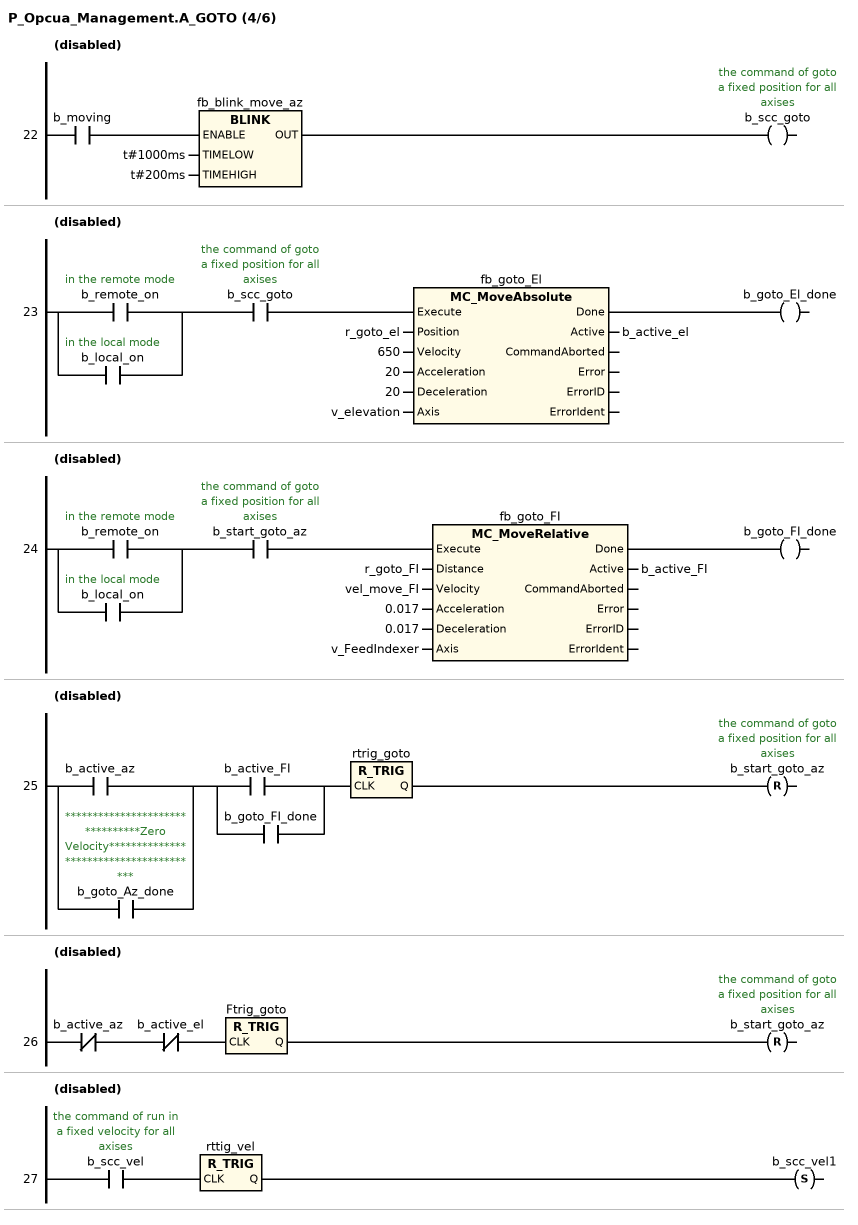
// NETWORK 22 (disabled)
//   b_scc_goto: the command of goto a fixed position for all axises
// fb_blink_move_az(ENABLE := b_moving, TIMELOW := t#1000ms, TIMEHIGH := t#200ms); // BLINK
// b_scc_goto := fb_blink_move_az.OUT;

// NETWORK 23 (disabled)
//   b_remote_on: in the remote mode
//   b_local_on: in the local mode
//   b_scc_goto: the command of goto a fixed position for all axises
//   v_elevation: Virtual axis "v_elevation" with axis number 8
// fb_goto_El(
//     Execute := (b_remote_on OR b_local_on) AND b_scc_goto,
//     Position := r_goto_el,
//     Velocity := 650,
//     Acceleration := 20,
//     Deceleration := 20,
//     Axis := v_elevation,
//     Active => b_active_el); // MC_MoveAbsolute
// b_goto_El_done := fb_goto_El.Done;

// NETWORK 24 (disabled)
//   b_remote_on: in the remote mode
//   b_local_on: in the local mode
//   b_start_goto_az: the command of goto a fixed position for all axises
//   v_FeedIndexer: Virtual axis "v_polarization" with axis number 9
// fb_goto_FI(
//     Execute := (b_remote_on OR b_local_on) AND b_start_goto_az,
//     Distance := r_goto_FI,
//     Velocity := vel_move_FI,
//     Acceleration := 0.017,
//     Deceleration := 0.017,
//     Axis := v_FeedIndexer,
//     Active => b_active_FI); // MC_MoveRelative
// b_goto_FI_done := fb_goto_FI.Done;

// NETWORK 25 (disabled)
//   b_goto_Az_done: ********************************Zero Velocity***************************************
//   b_start_goto_az: the command of goto a fixed position for all axises
// rtrig_goto(CLK := (b_active_az OR b_goto_Az_done) AND (b_active_FI OR b_goto_FI_done)); // R_TRIG
// b_start_goto_az R= rtrig_goto.Q;

// NETWORK 26 (disabled)
//   b_start_goto_az: the command of goto a fixed position for all axises
// Ftrig_goto(CLK := NOT b_active_az AND NOT b_active_el); // R_TRIG
// b_start_goto_az R= Ftrig_goto.Q;

// NETWORK 27 (disabled)
//   b_scc_vel: the command of run in a fixed velocity for all axises
// rttig_vel(CLK := b_scc_vel); // R_TRIG
// b_scc_vel1 S= rttig_vel.Q;

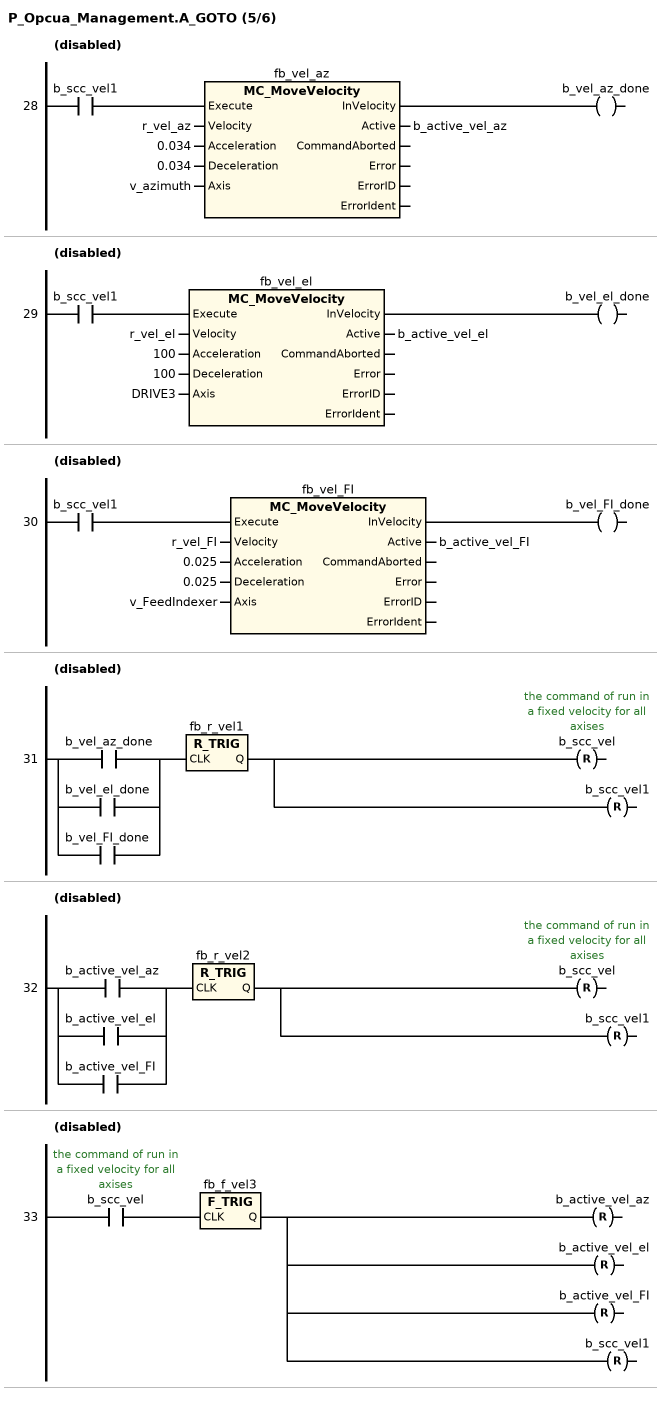
// NETWORK 28 (disabled)
//   r_vel_az: ************vel*************
//   v_azimuth: Virtual axis "v_azimuth" with axis number 7
// fb_vel_az(
//     Execute := b_scc_vel1,
//     Velocity := r_vel_az,
//     Acceleration := 0.034,
//     Deceleration := 0.034,
//     Axis := v_azimuth,
//     Active => b_active_vel_az); // MC_MoveVelocity
// b_vel_az_done := fb_vel_az.InVelocity;

// NETWORK 29 (disabled)
//   DRIVE3: Virtual axis "v_elevation" with axis number 8
// fb_vel_el(
//     Execute := b_scc_vel1,
//     Velocity := r_vel_el,
//     Acceleration := 100,
//     Deceleration := 100,
//     Axis := DRIVE3,
//     Active => b_active_vel_el); // MC_MoveVelocity
// b_vel_el_done := fb_vel_el.InVelocity;

// NETWORK 30 (disabled)
//   v_FeedIndexer: Virtual axis "v_polarization" with axis number 9
// fb_vel_FI(
//     Execute := b_scc_vel1,
//     Velocity := r_vel_FI,
//     Acceleration := 0.025,
//     Deceleration := 0.025,
//     Axis := v_FeedIndexer,
//     Active => b_active_vel_FI); // MC_MoveVelocity
// b_vel_FI_done := fb_vel_FI.InVelocity;

// NETWORK 31 (disabled)
//   b_scc_vel: the command of run in a fixed velocity for all axises
// fb_r_vel1(CLK := b_vel_az_done OR b_vel_el_done OR b_vel_FI_done); // R_TRIG
// b_scc_vel R= fb_r_vel1.Q;
// b_scc_vel1 R= fb_r_vel1.Q;

// NETWORK 32 (disabled)
//   b_scc_vel: the command of run in a fixed velocity for all axises
// fb_r_vel2(CLK := b_active_vel_az OR b_active_vel_el OR b_active_vel_FI); // R_TRIG
// b_scc_vel R= fb_r_vel2.Q;
// b_scc_vel1 R= fb_r_vel2.Q;

// NETWORK 33 (disabled)
//   b_scc_vel: the command of run in a fixed velocity for all axises
// fb_f_vel3(CLK := b_scc_vel); // F_TRIG
// b_active_vel_az R= fb_f_vel3.Q;
// b_active_vel_el R= fb_f_vel3.Q;
// b_active_vel_FI R= fb_f_vel3.Q;
// b_scc_vel1 R= fb_f_vel3.Q;

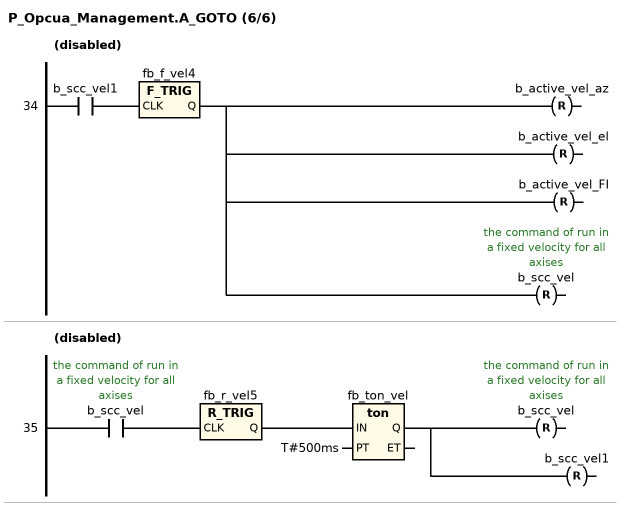
// NETWORK 34 (disabled)
//   b_scc_vel: the command of run in a fixed velocity for all axises
// fb_f_vel4(CLK := b_scc_vel1); // F_TRIG
// b_active_vel_az R= fb_f_vel4.Q;
// b_active_vel_el R= fb_f_vel4.Q;
// b_active_vel_FI R= fb_f_vel4.Q;
// b_scc_vel R= fb_f_vel4.Q;

// NETWORK 35 (disabled)
//   b_scc_vel: the command of run in a fixed velocity for all axises
// fb_r_vel5(CLK := b_scc_vel); // R_TRIG
// fb_ton_vel(IN := fb_r_vel5.Q, PT := T#500ms); // ton
// b_scc_vel R= fb_ton_vel.Q;
// b_scc_vel1 R= fb_ton_vel.Q;
END_ACTION

ACTION A_CLR_ERR:
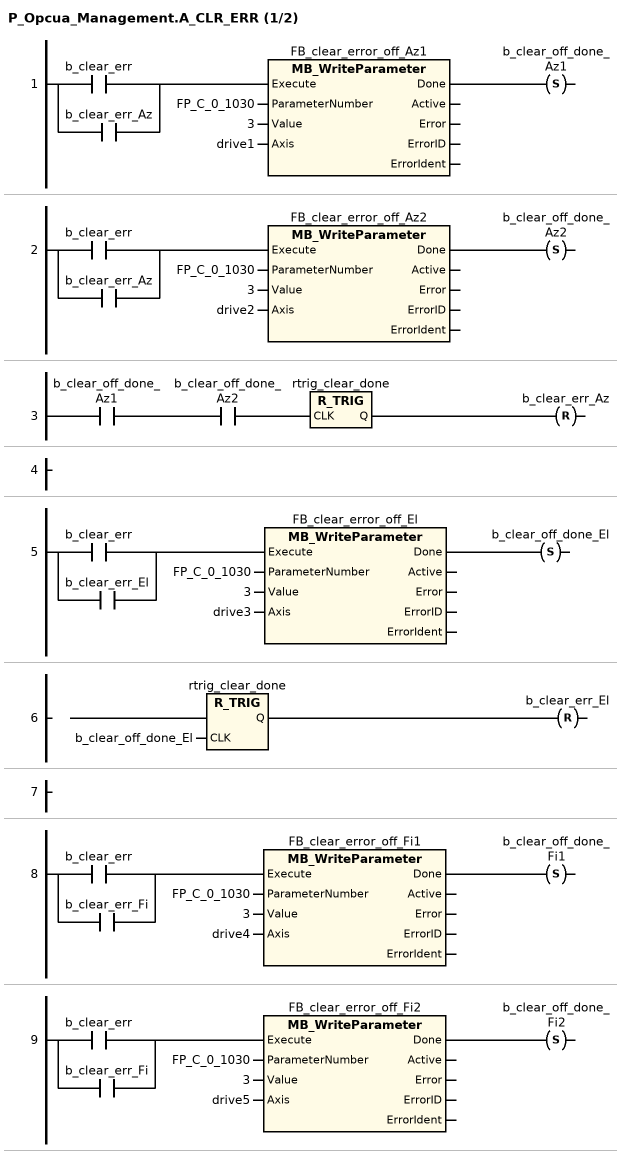
// NETWORK 1
//   FP_C_0_1030: Command: Clear all control errors
//   drive1: Real axis "Drive1" with axis number 1
FB_clear_error_off_Az1(
    Execute := b_clear_err OR b_clear_err_Az,
    ParameterNumber := FP_C_0_1030,
    Value := 3,
    Axis := drive1); // MB_WriteParameter
b_clear_off_done_Az1 S= FB_clear_error_off_Az1.Done;

// NETWORK 2
//   FP_C_0_1030: Command: Clear all control errors
//   drive2: Real axis "Drive1" with axis number 1
FB_clear_error_off_Az2(
    Execute := b_clear_err OR b_clear_err_Az,
    ParameterNumber := FP_C_0_1030,
    Value := 3,
    Axis := drive2); // MB_WriteParameter
b_clear_off_done_Az2 S= FB_clear_error_off_Az2.Done;

// NETWORK 3
rtrig_clear_done(CLK := b_clear_off_done_Az1 AND b_clear_off_done_Az2); // R_TRIG
b_clear_err_Az R= rtrig_clear_done.Q;

// NETWORK 4

// NETWORK 5
//   FP_C_0_1030: Command: Clear all control errors
//   drive3: Real axis "Drive1" with axis number 1
FB_clear_error_off_El(
    Execute := b_clear_err OR b_clear_err_El,
    ParameterNumber := FP_C_0_1030,
    Value := 3,
    Axis := drive3); // MB_WriteParameter
b_clear_off_done_El S= FB_clear_error_off_El.Done;

// NETWORK 6
rtrig_clear_done(CLK := b_clear_off_done_El); // R_TRIG
b_clear_err_El R= rtrig_clear_done.Q;

// NETWORK 7

// NETWORK 8
//   FP_C_0_1030: Command: Clear all control errors
//   drive4: Real axis "Drive1" with axis number 1
FB_clear_error_off_Fi1(
    Execute := b_clear_err OR b_clear_err_Fi,
    ParameterNumber := FP_C_0_1030,
    Value := 3,
    Axis := drive4); // MB_WriteParameter
b_clear_off_done_Fi1 S= FB_clear_error_off_Fi1.Done;

// NETWORK 9
//   FP_C_0_1030: Command: Clear all control errors
//   drive5: Real axis "Drive1" with axis number 1
FB_clear_error_off_Fi2(
    Execute := b_clear_err OR b_clear_err_Fi,
    ParameterNumber := FP_C_0_1030,
    Value := 3,
    Axis := drive5); // MB_WriteParameter
b_clear_off_done_Fi2 S= FB_clear_error_off_Fi2.Done;

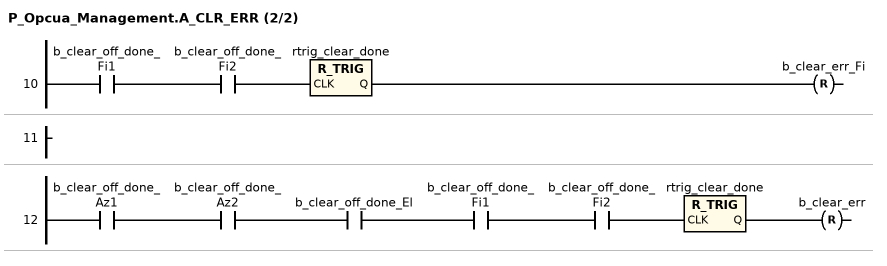
// NETWORK 10
rtrig_clear_done(CLK := b_clear_off_done_Fi1 AND b_clear_off_done_Fi2); // R_TRIG
b_clear_err_Fi R= rtrig_clear_done.Q;

// NETWORK 11

// NETWORK 12
rtrig_clear_done(CLK := b_clear_off_done_Az1 AND b_clear_off_done_Az2 AND b_clear_off_done_El AND b_clear_off_done_Fi1 AND b_clear_off_done_Fi2); // R_TRIG
b_clear_err R= rtrig_clear_done.Q;
END_ACTION

END_PROGRAM

// IndraMotionMlc1/Application/POUs/OPCUA/OPCUA_Node/P_Opcua_Tracking
{attribute 'linkalways'}
PROGRAM P_Opcua_Tracking
VAR_INPUT
	
	i_length: UINT;
	tai: ARRAY [1..1000] OF LREAL;
	Az: ARRAY [1..1000] OF LREAL;
	El: ARRAY [1..1000] OF LREAL;
	
END_VAR

VAR
	index: UINT; // Index used for addressing points in the tracking data arrays. 
	
	IL_LowPass_OnSource: IL_StateVariableType01;
	b_test: BOOL;
	
END_VAR


// Switch track on if the starttime has been reached
IF b_track_start AND (lr_track_start_time <= Time_cds.Status.TAIoffset) THEN 
	b_track_on:=1;
	b_track_start:=0;
END_IF

//IF i_length>0 THEN  // Load table into stack 
	
	
//END_IF

// Calculate whether the dish is on source. 

IF b_track_on THEN 
	IF  tracking.status.OnSourceDev <= Tracking.Status.OnSourceThreshold THEN 
		Management.Status.OnSource:=1;
	ELSE
		Management.Status.OnSource:=0;	
	END_IF
ELSE
	Management.Status.OnSource:=0;
END_IF

//Tracking.Status.act_statOffset_value_El  Updated in P_Track_cubic
//Tracking.Status.act_statOffset_value_Xel Updated in P_Track_cubic
//Tracking.Status.OnSourceDev              Updated in P_Track_cubic
//Tracking.Status.OnSourceThreshold        Updated in SetOnSourceThreshold
//Tracking.Status.p_desired_Az;            Updated in P_Track_cubic
//Tracking.Status.p_desired_El;            Updated in P_Track_cubic
//Tracking.Status.ThresholdTimePeriod      Updated in SetOnSourceThreshold
IF Management.Status.DscState=DscStatetype.Standby OR Management.Status.DscState=DscStatetype.Standstill OR Management.Status.DscState=DscStatetype.Slew OR Management.Status.DscState=DscStatetype.Track THEN 
	Tracking.Status.tr_initOk:=1;
ELSE 
	Tracking.Status.tr_initOk:=0;
END_IF

Tracking.Status.tr_obj_valid:= Tracking.TableStatus.pts_DataValid;
Tracking.Status.tr_selPoly:= 0;

IF Tracking.TableStatus.pts_DataValid THEN
	Tracking.Status.tr_TimeRemaining:= ABS(track_table[i_End].TAIoffset - track_table[i_Start].TAIoffset);
ELSE
	Tracking.Status.tr_TimeRemaining:=0;
END_IF

IF (track_table[i_End].TAIoffset)>(Time_cds.Status.TAIoffset+600) THEN  // Minimum of 10min track data available . 
	Tracking.Status.tr_valid:=1;
ELSE
	Tracking.Status.tr_valid:=0;
END_IF

Tracking.TableStatus.act_pt_act_index := INT_TO_UINT(i_Start);
Tracking.TableStatus.act_pt_end_index := INT_TO_UINT(i_End);
Tracking.TableStatus.act_pt_value_Az:= track_table[i_Start].Azimuth;
Tracking.TableStatus.act_pt_value_El:= track_table[i_Start].Elevation;
//Tracking.TableStatus.LastLoadMode; Updated in TrackloadTable
IF i_num_stack_left > 10 THEN
	Tracking.TableStatus.pts_Completed:=0; 
	ELSE
	Tracking.TableStatus.pts_Completed:=1;
END_IF
IF Tracking.TableStatus.pts_Completed THEN 
	Tracking.TableStatus.pts_DataValid:=0; // Once a track is finnished then there is no valid data to trck with. 
END_IF
Tracking.TableStatus.pts_Err:=0; 
//Tracking.TableStatus.pts_Interpol;  Updated in Track Start
Tracking.TableStatus.pts_InterpolError:=0;  // Don't have code for detecting interpolaor errors yet
Tracking.TableStatus.pts_Running:=b_track_on;
Tracking.TableStatus.pts_StartPos:=b_track_on;

IF i_num_stack_left<=60 AND i_num_stack_left >= 70 THEN
	Tracking.TableStatus.pts_TableAlmostFull:=1;
ELSE 
	Tracking.TableStatus.pts_TableAlmostFull:=0;
END_IF

P_Opcua_Tracking.A_Utils();

ACTION A_Utils:
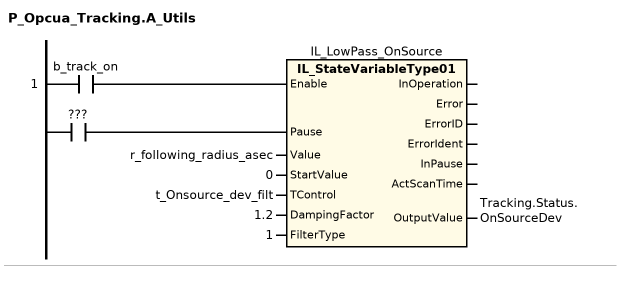
// NETWORK 1
IL_LowPass_OnSource(
    Enable := b_track_on,
    Value := r_following_radius_asec,
    StartValue := 0,
    TControl := t_Onsource_dev_filt,
    DampingFactor := 1.2,
    FilterType := 1,
    OutputValue => Tracking.Status.OnSourceDev); // IL_StateVariableType01
END_ACTION

END_PROGRAM

// IndraMotionMlc1/Application/POUs/OPCUA/OPCUA_Node/P_Opcua_Pointing
PROGRAM P_Opcua_Pointing
VAR
	TiltTemp_mV_1: LREAL;
	lr_one_x_off: LREAL;
	lr_one_y_off: LREAL;
	TiltTemp_mV_2: LREAL;
	lr_two_x_off: LREAL;
	lr_two_y_off: LREAL;
	IL_LowPass_Tilt_one_x: IL_StateVariableType01;
	IL_LowPass_Tilt_one_y: IL_StateVariableType01;
	IL_LowPass_Tilt_two_x: IL_StateVariableType01;
	IL_LowPass_Tilt_two_y: IL_StateVariableType01;
	t_one_x_filt_dt: TIME;
	t_one_y_filt_dt: TIME;
	t_two_x_filt_dt: TIME;
	t_two_y_filt_dt: TIME;
	b_tilt_filt_on: BOOL:= 1;
	RunOnce:Bool:=True;
END_VAR

Pointing();
(*****Data*****)
IF RunOnce THEN
	Pointing.StaticPmParameters:=StaticPmParametersSave;
	Pointing.TiltmeterParameters:=TiltmeterParametersSave;
	Pointing.AmbTempParameters:= AmbTempParametersSave;
	RunOnce:=FALSE; 
END_IF

(****************** Tilt Sensor **************************************)
// Tilt sensor one
Pointing.Status.TiltTemp_One := TiltTemp_mV_1*0.1;

lr_one_x_off:= (Pointing.TiltmeterParameters.One.x_zero+Pointing.TiltmeterParameters.One.x_zeroTC*Pointing.Status.TiltTemp_One)+
(Pointing.TiltmeterParameters.One.x_off+Pointing.TiltmeterParameters.One.x_offTC*Pointing.Status.TiltTemp_One);
lr_one_y_off:=(Pointing.TiltmeterParameters.One.y_zero+Pointing.TiltmeterParameters.One.y_zeroTC*Pointing.Status.TiltTemp_One)+
(Pointing.TiltmeterParameters.One.y_off+Pointing.TiltmeterParameters.One.y_offTC*Pointing.Status.TiltTemp_One);

Pointing.Status.TiltXArcsec_One:= Pointing.Status.TiltXRaw_mV_One*(Pointing.TiltmeterParameters.One.x_scale+Pointing.TiltmeterParameters.One.x_scaleTC*Pointing.Status.TiltTemp_One)+Pointing.TiltmeterParameters.One.x_off;
Pointing.Status.TiltYArcsec_One:= Pointing.Status.TiltYRaw_mV_One*(Pointing.TiltmeterParameters.One.y_scale+Pointing.TiltmeterParameters.One.y_scaleTC*Pointing.Status.TiltTemp_One)+Pointing.TiltmeterParameters.One.y_off;
t_one_x_filt_dt:= TO_TIME(Pointing.TiltmeterParameters.One.x_filt_dt*1000); //convert to milliseconds and TIME type.
t_one_y_filt_dt:= TO_TIME(Pointing.TiltmeterParameters.One.y_filt_dt*1000);

// Tilt Sensor Two
Pointing.Status.TiltTemp_Two := TiltTemp_mV_2*0.1;

lr_two_x_off:= (Pointing.TiltmeterParameters.Two.x_zero+Pointing.TiltmeterParameters.Two.x_zeroTC*Pointing.Status.TiltTemp_Two)+
(Pointing.TiltmeterParameters.Two.x_off+Pointing.TiltmeterParameters.Two.x_offTC*Pointing.Status.TiltTemp_Two);
lr_two_y_off:=(Pointing.TiltmeterParameters.Two.y_zero+Pointing.TiltmeterParameters.Two.y_zeroTC*Pointing.Status.TiltTemp_Two)+
(Pointing.TiltmeterParameters.Two.y_off+Pointing.TiltmeterParameters.Two.y_offTC*Pointing.Status.TiltTemp_Two);

Pointing.Status.TiltXArcsec_Two:= Pointing.Status.TiltXRaw_mV_Two*(Pointing.TiltmeterParameters.Two.x_scale+Pointing.TiltmeterParameters.Two.x_scaleTC*Pointing.Status.TiltTemp_Two)+Pointing.TiltmeterParameters.Two.x_off;
Pointing.Status.TiltYArcsec_Two:= Pointing.Status.TiltYRaw_mV_Two*(Pointing.TiltmeterParameters.Two.y_scale+Pointing.TiltmeterParameters.Two.y_scaleTC*Pointing.Status.TiltTemp_Two)+Pointing.TiltmeterParameters.Two.y_off;
t_two_x_filt_dt:= TO_TIME(Pointing.TiltmeterParameters.Two.x_filt_dt*1000); //convert to milliseconds and TIME type.
t_two_y_filt_dt:= TO_TIME(Pointing.TiltmeterParameters.Two.y_filt_dt*1000);

// Total point corrections

Pointing.Status.TotalPointCorr_Az:= Pointing.Status.StaticPmCorrVal_Az + Pointing.Status.TiltCorrVal_Az + Pointing.Status.AmbTempCorrVal_Az;
Pointing.Status.TotalPointCorr_El:= Pointing.Status.StaticPmCorrVal_El + Pointing.Status.TiltCorrVal_El + Pointing.Status.AmbTempCorrVal_El;

Pointing.Status.ActAmbTemp_East:= Pedestal_temp_1;  // These need to be checked
Pointing.Status.ActAmbTemp_South:= Pedestal_temp_2;;
Pointing.Status.ActAmbTemp_West:= Pedestal_temp_3;
//Pointing.Status.AmbTempCorrActive
//Pointing.Status.AmbTempCorrVal_Az
//Pointing.Status.AmbTempCorrVal_El
//Pointing.Status.BandForCorr
//Pointing.Status.StaticCorrActive
//Pointing.Status.StaticPmCorrVal_Az
//Pointing.Status.StaticPmCorrVal_El
//Pointing.Status.TiltCorrActive
//Pointing.Status.TiltCorrVal_Az
//Pointing.Status.TiltCorrVal_El
//Pointing.Status.TiltOne_On
//Pointing.Status.TiltTemp_One
//Pointing.Status.TiltTemp_Two
//Pointing.Status.TotalPointCorr_Az
//Pointing.Status.TotalPointCorr_El

ACTION A_Utils:
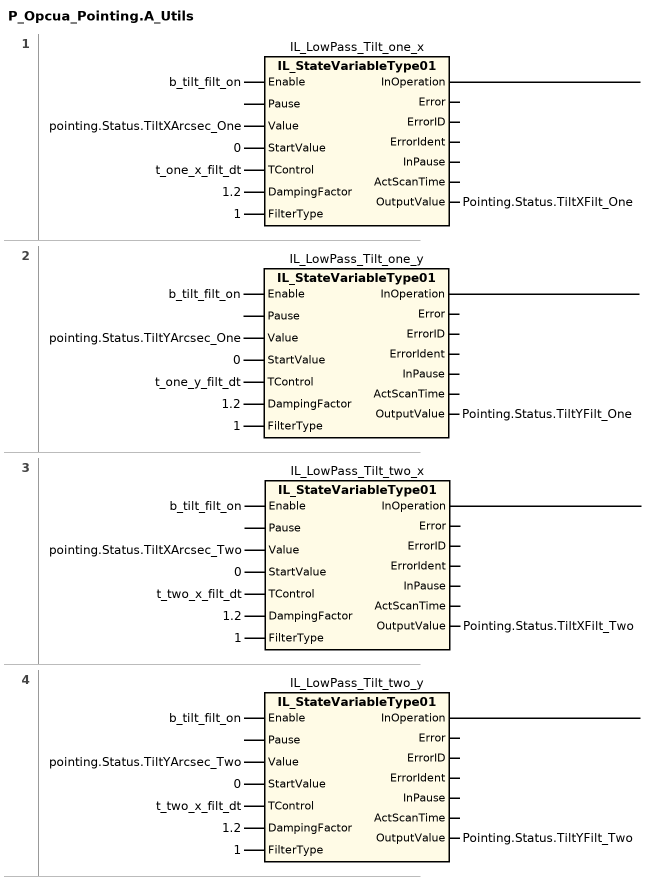
// NETWORK 1
IL_LowPass_Tilt_one_x(
    Enable := b_tilt_filt_on,
    Value := pointing.Status.TiltXArcsec_One,
    StartValue := 0,
    TControl := t_one_x_filt_dt,
    DampingFactor := 1.2,
    FilterType := 1,
    OutputValue => Pointing.Status.TiltXFilt_One); // IL_StateVariableType01

// NETWORK 2
IL_LowPass_Tilt_one_y(
    Enable := b_tilt_filt_on,
    Value := pointing.Status.TiltYArcsec_One,
    StartValue := 0,
    TControl := t_one_y_filt_dt,
    DampingFactor := 1.2,
    FilterType := 1,
    OutputValue => Pointing.Status.TiltYFilt_One); // IL_StateVariableType01

// NETWORK 3
IL_LowPass_Tilt_two_x(
    Enable := b_tilt_filt_on,
    Value := pointing.Status.TiltXArcsec_Two,
    StartValue := 0,
    TControl := t_two_x_filt_dt,
    DampingFactor := 1.2,
    FilterType := 1,
    OutputValue => Pointing.Status.TiltXFilt_Two); // IL_StateVariableType01

// NETWORK 4
IL_LowPass_Tilt_two_y(
    Enable := b_tilt_filt_on,
    Value := pointing.Status.TiltYArcsec_Two,
    StartValue := 0,
    TControl := t_two_x_filt_dt,
    DampingFactor := 1.2,
    FilterType := 1,
    OutputValue => Pointing.Status.TiltYFilt_Two); // IL_StateVariableType01
END_ACTION

END_PROGRAM

// IndraMotionMlc1/Application/POUs/Motion/Test_move
PROGRAM Test_move
VAR
	b_power: BOOL;
	b_enable_az1: BOOL;
	fb_enable_az1: MC_Power;
	b_enable_az1_done: BOOL;
	b_vel_az1: BOOL;
	fb_vel_az1: MC_MoveVelocity;
	vel_az1: REAL;
	b_enable_az2: BOOL;
	fb_enable_az2: MC_Power;
	b_enable_az2_done: BOOL;
	b_vel_az2: BOOL;
	vel_az2: REAL;
	fb_vel_az2: MC_MoveVelocity;
	b_enable_el1: BOOL;
	fb_enable_el1: MC_Power;
	b_enable_el1_done: BOOL;
	b_vel_el1: BOOL;
	vel_el1: REAL;
	fb_vel_el1: MC_MoveVelocity;
	b_vel_el2: BOOL;
	fb_vel_el2: MC_MoveVelocity;
	vel_el2: REAL;
	b_enable_el2: BOOL;
	fb_enable_el2: MC_Power;
	b_enable_FI1: BOOL;
	fb_enable_FI1: MC_Power;
	b_enable_el2_done: BOOL;
	b_enable_FI1_done: BOOL;
	b_vel_FI1: BOOL;
	fb_vel_FI1: MC_MoveVelocity;
	vel_FI1: REAL;
	b_enable_FI2: BOOL;
	fb_enable_FI2: MC_Power;
	b_enable_FI2_done: BOOL;
	b_vel_FI2: BOOL;
	vel_FI2: REAL;
	fb_vel_FI2: MC_MoveVelocity;
	b_torque_4: BOOL;
	b_torque_el2: BOOL;
	fb_torque_el2: MC_TorqueControl;
	b_torque_el2_done: BOOL;
	b_torque_az2: BOOL;
	fb_torque_az2: MC_TorqueControl;
	b_torque_az2_done: BOOL;
	fb_pos_az1: MC_MoveAbsolute;
	b_pos_az1: BOOL;
	pos_az1: REAL;
	b_stop_az: BOOL;
	fb_stop_AZ: MC_Stop;
	b_stop_el: BOOL;
	fb_stop_el: MC_Stop;
	b_pos_el1: BOOL;
	pos_el1: REAL;
	fb_pos_el1: MC_MoveAbsolute;
	b_pos_FI1: BOOL;
	pos_FI1: REAL;
	fb_pos_FI1: MC_MoveAbsolute;
	b_vel_1: BOOL;
	vel_1: REAL;
	fb_vel_1: MC_MoveVelocity;
	test_home_1: BOOL;
	fb_test_home: MB_Home;
	b_homeswitch_1: BOOL;
	b_torque_FI2: BOOL;
	fb_torque_FI2: MC_TorqueControl;
	b_torque_FI2_done: BOOL;
	b_touque_1: BOOL;
	fb_torque_az1: MC_TorqueControl;
	b_torque_az1_done: BOOL;
	torque_1: REAL;
	b_touque_3: BOOL;
	torque_3: REAL;
	fb_torque_el3: MC_TorqueControl;
END_VAR

(*IF r_pos_az>270.5 OR  r_pos_az<-270.5 THEN
			b_SCC_enable_on:=FALSE;
			b_SCC_enable_off:=TRUE; 
END_IF
*)




//axisdata[7].rActualPosition_i;
//test_move.power_move(); Commented out to prevent process using up resources.

ACTION power_move:
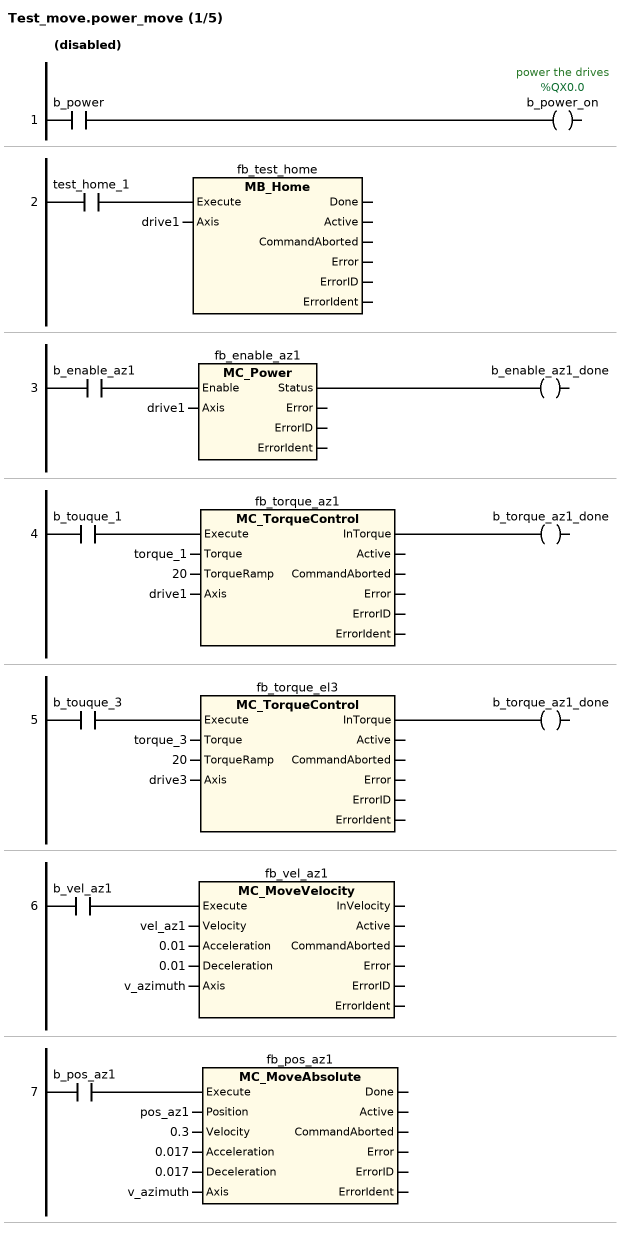
// NETWORK 1 (disabled)
//   b_power_on: power the drives | AT %QX0.0
// b_power_on := b_power;

// NETWORK 2
//   drive1: Real axis "Drive1" with axis number 1
fb_test_home(Execute := test_home_1, Axis := drive1); // MB_Home

// NETWORK 3
//   drive1: Real axis "Drive1" with axis number 1
fb_enable_az1(Enable := b_enable_az1, Axis := drive1); // MC_Power
b_enable_az1_done := fb_enable_az1.Status;

// NETWORK 4
//   drive1: Real axis "Drive4" with axis number 4
fb_torque_az1(Execute := b_touque_1, Torque := torque_1, TorqueRamp := 20, Axis := drive1); // MC_TorqueControl
b_torque_az1_done := fb_torque_az1.InTorque;

// NETWORK 5
//   drive3: Real axis "Drive4" with axis number 4
fb_torque_el3(Execute := b_touque_3, Torque := torque_3, TorqueRamp := 20, Axis := drive3); // MC_TorqueControl
b_torque_az1_done := fb_torque_el3.InTorque;

// NETWORK 6
//   v_azimuth: Virtual axis "v_azimuth" with axis number 7
fb_vel_az1(
    Execute := b_vel_az1,
    Velocity := vel_az1,
    Acceleration := 0.01,
    Deceleration := 0.01,
    Axis := v_azimuth); // MC_MoveVelocity

// NETWORK 7
//   v_azimuth: Virtual axis "v_azimuth" with axis number 7
fb_pos_az1(
    Execute := b_pos_az1,
    Position := pos_az1,
    Velocity := 0.3,
    Acceleration := 0.017,
    Deceleration := 0.017,
    Axis := v_azimuth); // MC_MoveAbsolute

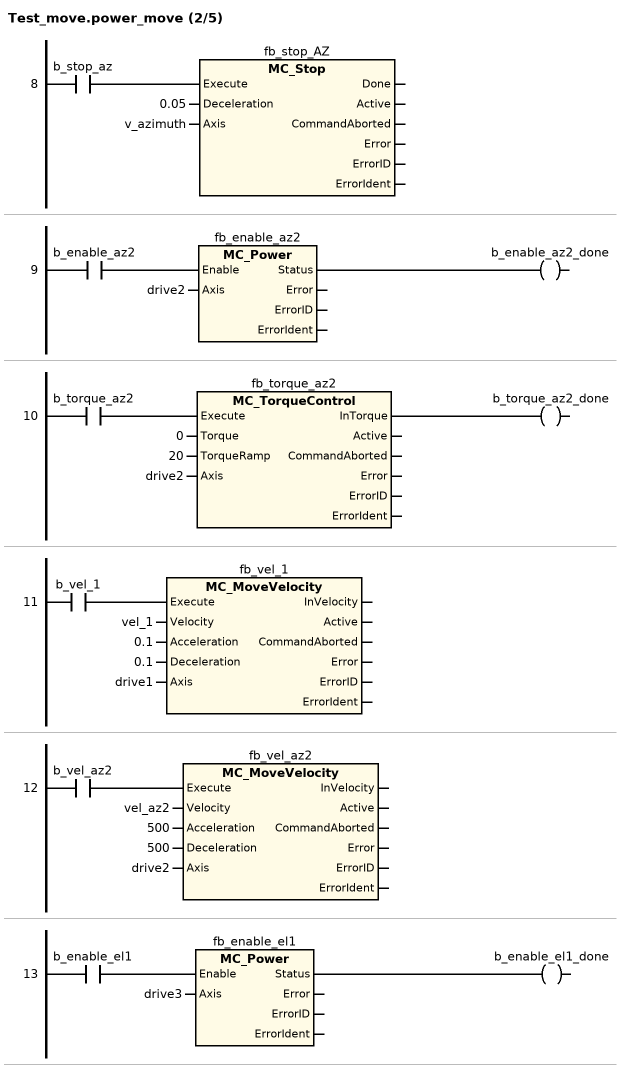
// NETWORK 8
//   v_azimuth: Virtual axis "v_azimuth" with axis number 7
fb_stop_AZ(Execute := b_stop_az, Deceleration := 0.05, Axis := v_azimuth); // MC_Stop

// NETWORK 9
//   drive2: Real axis "Drive2" with axis number 2
fb_enable_az2(Enable := b_enable_az2, Axis := drive2); // MC_Power
b_enable_az2_done := fb_enable_az2.Status;

// NETWORK 10
//   drive2: Real axis "Drive2" with axis number 2
fb_torque_az2(Execute := b_torque_az2, Torque := 0, TorqueRamp := 20, Axis := drive2); // MC_TorqueControl
b_torque_az2_done := fb_torque_az2.InTorque;

// NETWORK 11
//   drive1: Real axis "Drive1" with axis number 1
fb_vel_1(Execute := b_vel_1, Velocity := vel_1, Acceleration := 0.1, Deceleration := 0.1, Axis := drive1); // MC_MoveVelocity

// NETWORK 12
//   drive2: Real axis "Drive2" with axis number 2
fb_vel_az2(
    Execute := b_vel_az2,
    Velocity := vel_az2,
    Acceleration := 500,
    Deceleration := 500,
    Axis := drive2); // MC_MoveVelocity

// NETWORK 13
//   drive3: Real axis "Drive3" with axis number 3
fb_enable_el1(Enable := b_enable_el1, Axis := drive3); // MC_Power
b_enable_el1_done := fb_enable_el1.Status;

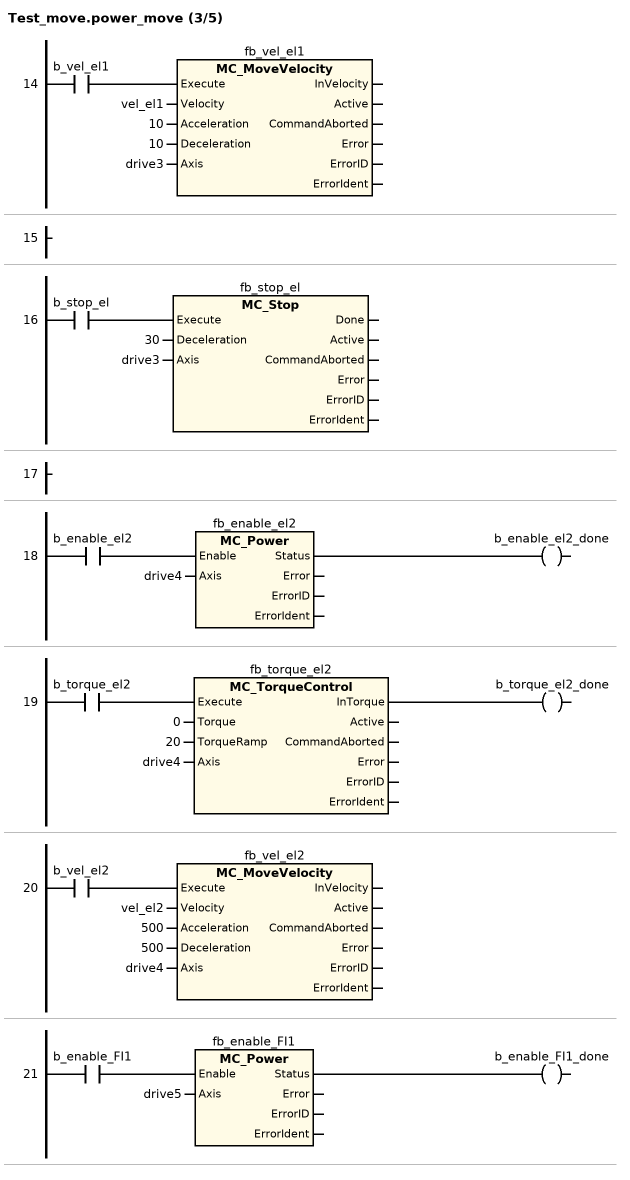
// NETWORK 14
//   drive3: Virtual axis "v_elevation" with axis number 8
fb_vel_el1(Execute := b_vel_el1, Velocity := vel_el1, Acceleration := 10, Deceleration := 10, Axis := drive3); // MC_MoveVelocity

// NETWORK 15

// NETWORK 16
//   drive3: Virtual axis "v_elevation" with axis number 8
fb_stop_el(Execute := b_stop_el, Deceleration := 30, Axis := drive3); // MC_Stop

// NETWORK 17

// NETWORK 18
//   drive4: Real axis "Drive4" with axis number 4
fb_enable_el2(Enable := b_enable_el2, Axis := drive4); // MC_Power
b_enable_el2_done := fb_enable_el2.Status;

// NETWORK 19
//   drive4: Real axis "Drive4" with axis number 4
fb_torque_el2(Execute := b_torque_el2, Torque := 0, TorqueRamp := 20, Axis := drive4); // MC_TorqueControl
b_torque_el2_done := fb_torque_el2.InTorque;

// NETWORK 20
//   drive4: Real axis "Drive4" with axis number 4
fb_vel_el2(
    Execute := b_vel_el2,
    Velocity := vel_el2,
    Acceleration := 500,
    Deceleration := 500,
    Axis := drive4); // MC_MoveVelocity

// NETWORK 21
//   drive5: Real axis "Drive5" with axis number 5
fb_enable_FI1(Enable := b_enable_FI1, Axis := drive5); // MC_Power
b_enable_FI1_done := fb_enable_FI1.Status;

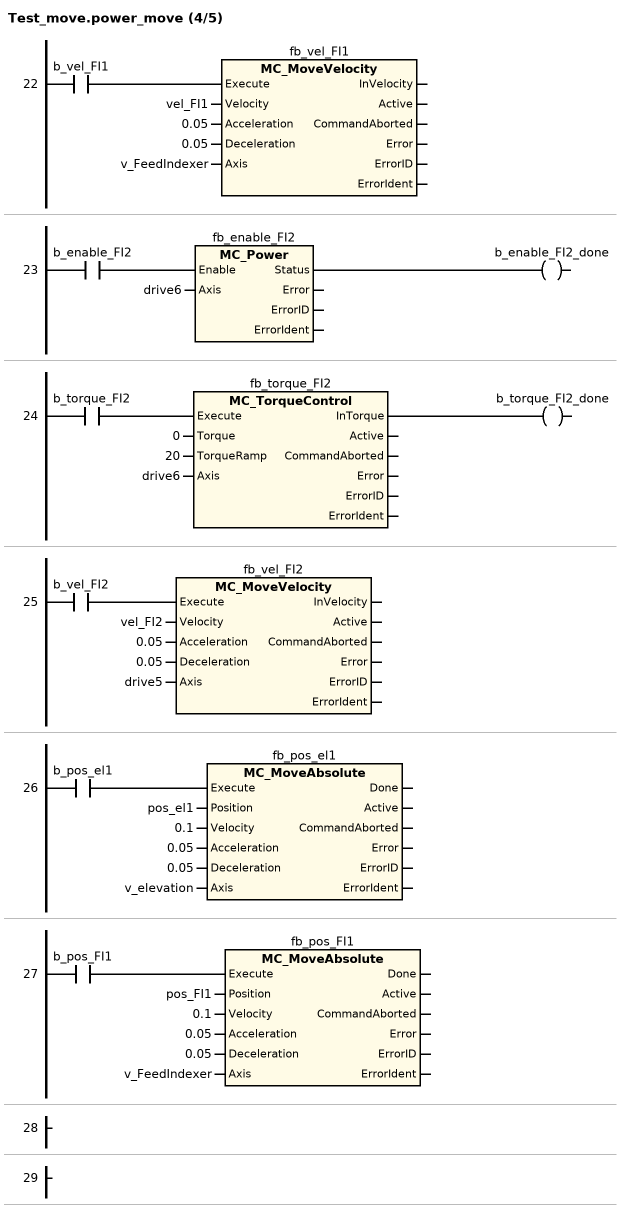
// NETWORK 22
//   v_FeedIndexer: Virtual axis "v_polarization" with axis number 9
fb_vel_FI1(
    Execute := b_vel_FI1,
    Velocity := vel_FI1,
    Acceleration := 0.05,
    Deceleration := 0.05,
    Axis := v_FeedIndexer); // MC_MoveVelocity

// NETWORK 23
//   drive6: Real axis "Drive6" with axis number 6
fb_enable_FI2(Enable := b_enable_FI2, Axis := drive6); // MC_Power
b_enable_FI2_done := fb_enable_FI2.Status;

// NETWORK 24
//   drive6: Real axis "Drive6" with axis number 6
fb_torque_FI2(Execute := b_torque_FI2, Torque := 0, TorqueRamp := 20, Axis := drive6); // MC_TorqueControl
b_torque_FI2_done := fb_torque_FI2.InTorque;

// NETWORK 25
//   drive5: Real axis "Drive5" with axis number 5
fb_vel_FI2(
    Execute := b_vel_FI2,
    Velocity := vel_FI2,
    Acceleration := 0.05,
    Deceleration := 0.05,
    Axis := drive5); // MC_MoveVelocity

// NETWORK 26
//   v_elevation: Virtual axis "v_elevation" with axis number 8
fb_pos_el1(
    Execute := b_pos_el1,
    Position := pos_el1,
    Velocity := 0.1,
    Acceleration := 0.05,
    Deceleration := 0.05,
    Axis := v_elevation); // MC_MoveAbsolute

// NETWORK 27
//   v_FeedIndexer: Virtual axis "v_polarization" with axis number 9
fb_pos_FI1(
    Execute := b_pos_FI1,
    Position := pos_FI1,
    Velocity := 0.1,
    Acceleration := 0.05,
    Deceleration := 0.05,
    Axis := v_FeedIndexer); // MC_MoveAbsolute

// NETWORK 28

// NETWORK 29

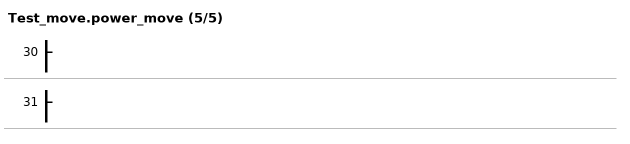
// NETWORK 30

// NETWORK 31
END_ACTION

END_PROGRAM

// IndraMotionMlc1/Application/POUs/Motion/PlcProg
PROGRAM PlcProg
VAR
	bVM_Enable: BOOL;
	rVM_Acc: REAL:=10.0;
	rVM_Dec: REAL:=10.0;
	rVM_Velocity: REAL:=3.0;
  rPhaseShift: REAL:=99.0;
	bVM_VelModeAck: BOOL;
	bVM_Standstill: BOOL;
	rVM_actVelocity: REAL;
END_VAR

//------------------------------------------------------------------------------------------------------
//--------------------- Call all required programs --> Imc and Axis Interface Update  ------------------  
//------------------------------------------------------------------------------------------------------
TE_AxisInterfaceType01Prog();
MB_ImcInterface();

IF TE_AxisInterfaceType01Prog.InitDone=FALSE THEN
	RETURN;
END_IF


//------------------------------------------------------------------------------------------------------
//----------------------------- Example for axis-access with AxisInterface ------------------------------  
//------------------------------------------------------------------------------------------------------

//----------------
// Axis-Command
//----------------
(*IF bRemoteOn_gb = FALSE THEN
 // arAxisCtrl_gb[MyVirtualAxis1.AxisNo].Admin._OpMode.b.MODE_VEL := bVM_Enable;
  IF bVM_Enable THEN
		arAxisCtrl_gb[MyVirtualAxis1.AxisNo].Admin._OpMode.en := ModeVel;
		arAxisCtrl_gb[MyVirtualAxis2.AxisNo].Admin._OpMode.en := ModeSyncPhase;
	ELSE
		arAxisCtrl_gb[MyVirtualAxis1.AxisNo].Admin._OpMode.en := ModeAb;
		arAxisCtrl_gb[MyVirtualAxis2.AxisNo].Admin._OpMode.en := ModeAb;
	END_IF
  arAxisCtrl_gb[MyVirtualAxis1.AxisNo].VelMode.Acceleration := rVM_Acc;
  arAxisCtrl_gb[MyVirtualAxis1.AxisNo].VelMode.Deceleration := rVM_Dec;
  arAxisCtrl_gb[MyVirtualAxis1.AxisNo].VelMode.Velocity := rVM_Velocity;
  arAxisCtrl_gb[MyVirtualAxis2.AxisNo].SyncMode.Master := MyVirtualAxis1;
  arAxisCtrl_gb[MyVirtualAxis2.AxisNo].SyncMode.PhaseShift := rPhaseShift;
END_IF
//----------------
// Axis-Status 
//----------------
bVM_VelModeAck := arAxisStatus_gb[MyVirtualAxis1.AxisNo].Admin.MODE_VEL;
IF (arAxisStatus_gb[MyVirtualAxis1.AxisNo].Admin.Active = TRUE) THEN
  // Pointer access only when axis is available -> avoid exceptions
  bVM_Standstill := arAxisStatus_gb[MyVirtualAxis1.AxisNo].PtrAxisData^.Axis_Standstill;
  rVM_actVelocity := arAxisStatus_gb[MyVirtualAxis1.AxisNo].PtrAxisData^.rActualVelocity_i;
END_IF
// Axis information can be evualated directly from AxisData-Array (same information at PtrAxisData^)
// AxisData[VM_Axis.AxisNo].Axis_Standstill;
// AxisData[VM_Axis.AxisNo].rActualVelocity_i;
*)

END_PROGRAM

// IndraMotionMlc1/Application/AxisInterface/TE_AxisInterfaceType01Prog
PROGRAM TE_AxisInterfaceType01Prog
(*#############################################################################################
  #############################################################################################  

   General Header   
  ---------------------------------------------------------------------------------------------  
   Shortdescription       : Cyclic execution of the Axis-Interface (POS, VEL and SYNC mode)
   Version                : see Version Function
   Name                   : DC-IA/EAM4 (KG)
   Date                   : see Version Function
   Company                : see Version Function
   Target                 : see Version Function
   Functional description : This program executes cyclic the axis interface FB for all axes.
                            The execution time of the axis interface FB is measured.
   Handling specials      : The global arrays of the axis-interface must be named arAxisCtrl_gb[]
                            and arAxisStatus_gb[]
  ---------------------------------------------------------------------------------------------  
    
   Additional Header   
  ---------------------------------------------------------------------------------------------  
  #############################################################################################  
  #############################################################################################*)
(*
                                     ******************
                                     *   DISCLAIMER   *
                                     ******************
   It is acknowledged that with regard to these software programs and program modules free of
   charge, Bosch Rexroth's usually practised, in-house test and release procedures have not 
   been accomplished. These software programs and program modules free of charge serve only as
   an example for possible applications.  They are intended as a help in order to obtain addi-
   tional experience regarding function, operation, performance and capacity of a maybe later 
   issued series release. Therefore Bosch Rexroth disclaims any liability and rejects to assume
   responsibility that these software programs or program modules, including any information 
   and data stored in those programs, are suitable for any intended use or that these programs
   will work without errors in any combination with the data processing environment. Providing
   you with these software programs shall neither constitute a claim for technical support nor
   for any other remedy for defects. Any claims for damages of any nature and for any legal
   reason arising from installing or using these software programs or program modules are ex-
   cluded, unless these damages was caused by Bosch Rexroth`s statutory representatives or em-
   ployees by wilful misconduct or by gross negligence or liability is compulsory in accordance
   with the German product liability law. In any case Bosch Rexroth`s liability for any conse-
   quential or incidental damages such as, but not limited to loss of profit, loss of pro-
   duction or loss of data is excluded.      
*)
(*---------------------------------------------------------------------------------------------*)
VAR_INPUT
  ClearError: BOOL;		// clear internal errors of the program
END_VAR
VAR_OUTPUT
  InitDone: BOOL;		// Init is done, AxisInterface is ready to operate
  Error: BOOL;			// internal error of the program
  ErrorID: ERROR_CODE;
  ErrorIdent: ERROR_STRUCT;
END_VAR
VAR CONSTANT
   STATE_FIRST_INIT       : UINT := 0;
   STATE_WAIT_FOR_PHASE2  : UINT := 1;
   STATE_INIT_P2          : UINT := 2;
   STATE_WAIT_FOR_PHASE3  : UINT := 3;
   STATE_INIT_P3          : UINT := 4;
   STATE_WAIT_FOR_PHASE4  : UINT := 5;
   STATE_WAIT_FOR_NOT_P4  : UINT := 6;
   STATE_PRG_ERROR        : UINT := 9;
   
   dwADD1_STATE_MACHINE_ERROR: DWORD := 16#00000006;
   dwADD2_STATE_MACHINE_ERROR: DWORD := 16#00000000;
   
END_VAR
VAR
    fbAxisInitAllAxis: TE_AxisInitAllAxisType01; //  basic init of arAxisCtrl structure 

    uiState                 : UINT := STATE_FIRST_INIT; // statemachine
	  // Flag that the inputs of the FB are set
	  bInitReferencesDone: BOOL; 
  
    fbAxis                    : ARRAY [1..uiMAX_AXIS_INDEX] OF TE_AxisInterface;
	  uiLoop                    : UINT := 1;
    uiAxisIdx                 : UINT; // axis index for the list without gaps
	  // time measurement
    udiStartTime              : UDINT;
    udiStopTime               : UDINT;
	  udiActCycleTime           : UDINT;
    stCyclesTime              : TE_PLC_CYCLES_TIME;
END_VAR

// -------------------------------------------------------------------------------- 
// state-machine: do the warmstart initialisation everytime we reach SERCOS phase 4 
// -------------------------------------------------------------------------------- 
CASE uiState OF

  STATE_FIRST_INIT:
    // ---------------------------------------------------------------------------------
    // Step: Done only once when PLC program starts.           
    // ---------------------------------------------------------------------------------
   	FOR uiLoop := 1 TO uiMAX_AXIS_INDEX DO
		 	fbAxis[uiLoop].mInitExtension(uiLoop);
		END_FOR
		bInitReferencesDone := TRUE; // Inputs are set, FB can be called	
    uiState := STATE_WAIT_FOR_PHASE2;
  
  STATE_WAIT_FOR_PHASE2:
    // --------------------------------------------------------------------------------- 
    // Step: Wait for SERCOS phase P2;                                                   
    // Done cyclic when we are in phases < 2                                             
    // --------------------------------------------------------------------------------- 
    IF (ImcStatus.Admin.ModeStatus_P2 = TRUE) THEN
      uiState := STATE_INIT_P2;
      InitDone := FALSE;      
		ELSIF( (ImcStatus.Admin.PwrUpModeAck = TRUE) AND (ImcStatus.Admin._OpModeAck > IMC_MODE_STATUS_P2) ) THEN
  	// E.g. PL program download in P4, go directly to P4
      uiState := STATE_INIT_P3;
      InitDone := FALSE;      
    END_IF
	
  STATE_INIT_P2:
    // --------------------------------------------------------------------------------- 
    // Step: Action actInitWarmStart. Done when reaching parameter mode.                 
    // --------------------------------------------------------------------------------- 
    actInitWarmStart();

  STATE_WAIT_FOR_PHASE3:
    // --------------------------------------------------------------------------------- 
    // Step: Wait for SERCOS phase P3;                 
    // Start Init once when reaching CP3                                   
    // ---------------------------------------------------------------------------------
    IF( ImcStatus.Admin._OpModeAck >= IMC_MODE_STATUS_P3 ) THEN
      uiState := STATE_INIT_P3;
      InitDone := FALSE;      
    END_IF


  STATE_INIT_P3:
    // --------------------------------------------------------------------------------- 
    // Step: Action actInitWarmStart. Done when reaching CP3                 
    // --------------------------------------------------------------------------------- 
    actInitWarmStart();

  STATE_WAIT_FOR_PHASE4:
    // --------------------------------------------------------------------------------- 
    // Step: Wait for SERCOS phase P4;                                                   
    // ---------------------------------------------------------------------------------
    IF( ImcStatus.Admin.ModeStatus_BB = TRUE ) THEN
      uiState := STATE_WAIT_FOR_NOT_P4;
    END_IF
    // Falling back into CP2 ? Return 
    IF (ImcStatus.Admin.ModeStatus_P2 = TRUE) THEN
      uiState := STATE_INIT_P2;
      InitDone := FALSE;      
    END_IF

  STATE_WAIT_FOR_NOT_P4:
    // --------------------------------------------------------------------------------- 
    // Step: Check SECROS phase changes from P4                                          
    // Done cyclic when we are in phase 4                                                
    // --------------------------------------------------------------------------------- 

    // Check if we have left phase 4 
    IF( (ImcStatus.Admin.ModeStatus_BB = FALSE) OR (InitDone = FALSE) ) THEN
      // We have left phase 4 -> re-init the axis interface 
      uiState := STATE_WAIT_FOR_PHASE4;
    END_IF
	
  STATE_PRG_ERROR:
    IF ClearError = TRUE THEN
      // clear error information
      Error := FALSE;
      InitDone := FALSE; // enforce a new init 
      uiState := STATE_WAIT_FOR_PHASE4;
    END_IF
	
  ELSE
	// -------------------------------------------- 
    // DEFAULT case -> Signal error !!!                      
    // -------------------------------------------- 
    Error := TRUE;
    // set error information
    ErrorID := STATE_MACHINE_ERROR;
    ErrorIdent.Table := F_RELATED_TABLE;
	  ErrorIdent.Additional1 := dwADD1_STATE_MACHINE_ERROR;
	  ErrorIdent.Additional2 := dwADD2_STATE_MACHINE_ERROR;
    uiState := STATE_PRG_ERROR; 

END_CASE

udiStartTime := IL_HighResTimeTick(TRUE); // latch starting time 

IF (InitDone AND bInitReferencesDone) THEN
  FOR uiLoop := 1 TO uiNofAxis_gb DO
    uiAxisIdx := arAxisIdx_gb[uiLoop];
		// comment the next line for performance optimisation, but then do no online-change!!!
		fbAxis[uiAxisIdx].mInitExtension(uiAxisIdx); // set inputs always to avoid online change problems  
    fbAxis[uiAxisIdx]( ); // call FB, inputs are already set....
  END_FOR
END_IF  

udiStopTime := IL_HighResTimeTick(TRUE); // latch end time 

// calculate actual runtime and store MIN and MAX 
udiActCycleTime := IL_HighResTimeDiff(udiStartTime,udiStopTime);

stCyclesTime.udiActualTime := udiActCycleTime;

IF (stCyclesTime.udiMaximumTime < udiActCycleTime) THEN
  stCyclesTime.udiMaximumTime := udiActCycleTime;
END_IF

IF (stCyclesTime.udiMinimumTime > udiActCycleTime) THEN
  stCyclestime.udiMinimumTime := udiActCycleTime;
END_IF

ACTION actInitWarmStart:
// --------------------------------------------------------------------------------- 
// Action actInitWarmStart: Done when reaching parameter mode (P2)                   
// and again when reaching operating mode (phase 4)             	             
// --------------------------------------------------------------------------------- 

// ############################################ 
// Step: Basic Init of arAxisCtrl_gb for all axes  
// ############################################ 
fbAxisInitAllAxis(
  Execute:= TRUE,
  ReadModuloValue:=TRUE,
  EnableCyclicScanning:=TRUE );

IF(fbAxisInitAllAxis.Error = TRUE) THEN
  // -------------------------------------------- 
  // Signal error !!!                      
  // -------------------------------------------- 
  Error := TRUE;
  // copy error information
  ErrorID := fbAxisInitAllAxis.ErrorID;
  ErrorIdent := fbAxisInitAllAxis.ErrorIdent;
  // reset FB 
  fbAxisinitAllAxis( Execute := FALSE );
  // go to error state
  uiState := STATE_PRG_ERROR; 
  
ELSIF(fbAxisInitAllAxis.Done = TRUE) THEN
  // -------------------------------------------- 
  // Signal init is finished                      
  // -------------------------------------------- 
  InitDone := TRUE; // Init is finished 
  // reset FB 
  fbAxisinitAllAxis( Execute := FALSE );
  

  // ---------------------------------------------------------------------------------
  // End of this state by increasing uiState (call from STATE_INIT_P2 or STATE_INIT_P4)                                          
  // ---------------------------------------------------------------------------------
  uiState := uiState + 1;
END_IF
END_ACTION

END_PROGRAM

// IndraMotionMlc1/Application/AxisInterface/TE_AxisInitAllAxisType01
(* Initialisation of the Axis-Interface (POS, VEL and SYNC mode)
  #############################################################################################
  #############################################################################################  

   General Header   
  ---------------------------------------------------------------------------------------------  
   Shortdescription       : Initialisation of the Axis-Interface (POS, VEL and SYNC mode)
   Version                : see Version Function
   Name                   : Dc-IA/EAM (KG,PoVa)
   Date                   : see Version Function
   Company                : see Version Function  
   Target                 : see Version Function
   Functional description : This functionblocks initialises the data structures for the
                            axis interface. All available axes (C-0-0484) are activated.
   Handling specials      : The global arrays of the axis-interface must be named arAxisCtrl_gb[]
                            and arAxisStatus_gb[]. The variables for the axis list without gaps 
                            must be named arAxisIdx_gb and uiNofAxis_gb. 
  ---------------------------------------------------------------------------------------------  
    
   Additional Header   
     The following structure elements are set by this function block:
      arAxisCtrl_gb[].Admin._OpMode.en = ModeAB
      arAxisCtrl_gb[].Admin.ClearError = FALSE      
      arAxisCtrl_gb[].Admin.LockInputChanges = FALSE       
      arAxisCtrl_gb[].Admin.SetAbsRef = FALSE      
      arAxisCtrl_gb[].Admin.Axis.CntrlNo = LOCAL_CNTRL;
      arAxisCtrl_gb[].Admin.Axis.AxisNo = AXIS_1 .. AXIS_n
      arAxisCtrl_gb[].PosMode.Adjust.Enable = FALSE       
      arAxisCtrl_gb[].VelMode.Adjust.Enable = FALSE       
      arAxisCtrl_gb[].SyncMode.AdjCamShaftDist.Enable = FALSE       
      arAxisCtrl_gb[].SyncMode.AdjFineadjust.Enable = FALSE         
      arAxisCtrl_gb[].SyncMode.AdjPhaseOffset.Enable = FALSE        
      arAxisCtrl_gb[].Comment = A-0-0002

      arAxisStatus_gb[].Active = TRUE for active axis ( C-0-0484 )
      arAxisStatus_gb[].Admin.AxisFeatures = set with value of A-0-0004 for all axis

    Only when ReadModuloValue = TRUE and the axis is rotatoric:
      arAxisCtrl_gb[iAxisNo].PosMode.Adjust.ModuloValue = A-0-0045
      arAxisCtrl_gb[iAxisNo].SyncMode.AdjPhaseOffset.ModuloValue = A-0-045
      arAxisCtrl_gb[iAxisNo].VelMode.Adjust.ModuloValue = 0
      arAxisCtrl_gb[iAxisNo].SyncMode.AdjCamShaftDist.ModuloValue = 0
      arAxisCtrl_gb[iAxisNo].SyncMode.AdjFineadjust.ModuloValue = 0

  ---------------------------------------------------------------------------------------------  
     
     
     
  ---------------------------------------------------------------------------------------------  

  #############################################################################################  
  #############################################################################################*)
(*
                                     ******************
                                     *   DISCLAIMER   *
                                     ******************
   It is acknowledged that with regard to these software programs and program modules free of
   charge, Bosch Rexroth's usually practised, in-house test and release procedures have not 
   been accomplished. These software programs and program modules free of charge serve only as
   an example for possible applications.  They are intended as a help in order to obtain addi-
   tional experience regarding function, operation, performance and capacity of a maybe later 
   issued series release. Therefore Bosch Rexroth disclaims any liability and rejects to assume
   responsibility that these software programs or program modules, including any information 
   and data stored in those programs, are suitable for any intended use or that these programs
   will work without errors in any combination with the data processing environment. Providing
   you with these software programs shall neither constitute a claim for technical support nor
   for any other remedy for defects. Any claims for damages of any nature and for any legal
   reason arising from installing or using these software programs or program modules are ex-
   cluded, unless these damages was caused by Bosch Rexroth`s statutory representatives or em-
   ployees by wilful misconduct or by gross negligence or liability is compulsory in accordance
   with the German product liability law. In any case Bosch Rexroth`s liability for any conse-
   quential or incidental damages such as, but not limited to loss of profit, loss of pro-
   duction or loss of data is excluded.      
*)
(*---------------------------------------------------------------------------------------------*)

FUNCTION_BLOCK TE_AxisInitAllAxisType01

VAR_INPUT
    Execute         : BOOL;            (* start execution with rising edge *)
    ReadModuloValue : BOOL := TRUE;    (* Read parameters A59 and A45 and write the modulo value
                                          for rotatoric axis to the adjustment structure of PosMode
                                          SyncMode.AdjPhaseOffset and set modulo value to 0 for all
                                          other adjusted values. Activate before "Execute" *)
    EnableCyclicScanning : BOOL := TRUE; (* Enable the cyclic check and transmission of changed
                                            inputs for the actual operating mode
                                            - relevant for the values in AxisCtrl with 
                                              "Note: cyclic checked AND transmitted on change" *)
END_VAR

VAR_OUTPUT
    {attribute 'analysis' := '-27'} // disable static code analysis rule 27, check of same names 
    Done        : BOOL := FALSE;       (* Is SET when FB has finished operation *)
    Active      : BOOL := FALSE;       (* Is SET when FB is active (not in idle mode) *)
    {attribute 'analysis' := '-27'} // disable static code analysis rule 27, check of same names 
    Error       : BOOL := FALSE;       (* ErrorFlag *)
    ErrorID     : ERROR_CODE;          (* Error identification, Errorcode *)
    ErrorIdent  : ERROR_STRUCT;        (* Error identification *)
END_VAR

VAR
    bOldExecute         : BOOL := FALSE;
    uiState             : UINT := 0;
    stDummyAxis         : AXIS_REF;
    arBuffer            : ARRAY [1..(MB_MAX_AXIS_NUMBER*2)] OF INT;
    fbReadListParaC484  : MB_ReadListParameter;
    uiAxisNo            : UINT   := 1;
    Axis                : AXIS_REF;
    fbAxisInitType01    : MB_AxisInitType01;
    uiLoop              : UINT;
END_VAR

VAR CONSTANT
   STATE_DO_NOTHING             : UINT := 0;
   STATE_READ_C484              : UINT := 1;
   STATE_CHK_AXIS               : UINT := 2;
   STATE_START_INIT             : UINT := 3;
	 STATE_ERROR									: UINT := 99;
END_VAR

(* Detect rising edge *)
IF( (Execute = TRUE) AND (bOldExecute = FALSE) ) THEN
     uiState := STATE_READ_C484;
END_IF

CASE uiState OF

    STATE_DO_NOTHING:
      IF( Execute = FALSE ) THEN
        (* RESET everything *)
        Done    := FALSE;
        Active  := FALSE;
        Error   := FALSE;
        uiAxisNo := 1;
      END_IF;

    STATE_READ_C484:
      (* ############################################### *)
      (* Step: Read C-0-0484 "Axes configuration list"   *)
      (* ############################################### *)

      fbReadListParaC484(
        Execute           := TRUE,
        ParameterNumber   := FP_C_0_0484,
        NoOfBytes         := SIZEOF(arBuffer),
        ValueAdr          := ADR(arBuffer),
        Axis              := stDummyAxis);

      IF ( fbReadListParaC484.Done = TRUE ) THEN
        (* reset FB *)
        fbReadListParaC484(
          Execute    := FALSE,
          Axis       := stDummyAxis);
        uiState := STATE_CHK_AXIS;
        uiAxisNo := 1;
        // reset list of all axes
        FOR uiLoop:=1 TO uiMAX_AXIS_INDEX DO
          arAxisIdx_gb[uiLoop] := 0;
				END_FOR
        uiNofAxis_gb := 0; // reset global axis counter 
      ELSIF ( fbReadListParaC484.Error = TRUE ) THEN
				Error := TRUE;
        ErrorID := fbReadListParaC484.ErrorID;
				ErrorIdent := fbReadListParaC484.ErrorIdent;
        (* reset FB *)
        fbReadListParaC484(
          Execute    := FALSE,
          Axis       := stDummyAxis);
        uiState := STATE_ERROR;
      END_IF

  STATE_CHK_AXIS:
    (* ############################################ *)
    (* Step: Check all configured axis              *)
    (* ############################################ *)
    IF ( uiAxisNo <= uiMAX_AXIS_INDEX ) THEN
      (* activate, when axis type not equal 0 *)
      IF ( arBuffer[2*uiAxisNo - 1] <> 0 ) THEN
        uiState      := STATE_START_INIT;
        Axis.AxisNo := UINT_TO_INT(uiAxisNo);
        Axis.CntrlNo := LOCAL_CNTRL;
        uiNofAxis_gb:=uiNofAxis_gb+1; // increase axes counter
        arAxisIdx_gb[uiNofAxis_gb] := uiAxisNo; // store the index in the lagless list 
      ELSE
        uiAxisNo := uiAxisNo + 1;
      END_IF

    ELSE
      Done    := TRUE;
      Active  := FALSE;
      uiState := STATE_DO_NOTHING;
    END_IF

  STATE_START_INIT:
    (* ############################################ *)
    (* Step: Initialize all configured axis         *)
    (* ############################################ *)

    (* call FB ML_AxisInitType01 -> initialize the axis *)
    fbAxisInitType01(
      Execute              := TRUE,
      ReadModuloValue      := ReadModuloValue,
      EnableCyclicScanning := EnableCyclicScanning,
      AdminCtrl            := arAxisCtrl_gb[uiAxisNo].Admin,
      PosModeCtrl          := arAxisCtrl_gb[uiAxisNo].PosMode,
      VelModeCtrl          := arAxisCtrl_gb[uiAxisNo].VelMode,
      SyncModeCtrl         := arAxisCtrl_gb[uiAxisNo].SyncMode,
      AxisDataPtrStatus    := arAxisStatus_gb[uiAxisNo].PtrAxisData,
      AdminStatus          := arAxisStatus_gb[uiAxisNo].Admin,
      DiagStatus           := arAxisStatus_gb[uiAxisNo].Diag,
      Axis                 := Axis);
    IF ( fbAxisInitType01.Error = TRUE ) THEN
      Error      := fbAxisInitType01.Error;
      ErrorID    := fbAxisInitType01.ErrorID;
      ErrorIdent := fbAxisInitType01.ErrorIdent;
 		  uiState    := STATE_ERROR;
    ELSIF ( fbAxisInitType01.Done = TRUE ) THEN
      (* restart ML_AxisInitType01 *)
      fbAxisInitType01(
        Execute            := FALSE,
        AdminCtrl          := arAxisCtrl_gb[uiAxisNo].Admin,
        PosModeCtrl        := arAxisCtrl_gb[uiAxisNo].PosMode,
        VelModeCtrl        := arAxisCtrl_gb[uiAxisNo].VelMode,
        SyncModeCtrl       := arAxisCtrl_gb[uiAxisNo].SyncMode,
        AxisDataPtrStatus  := arAxisStatus_gb[uiAxisNo].PtrAxisData,
        AdminStatus        := arAxisStatus_gb[uiAxisNo].Admin,
        DiagStatus         := arAxisStatus_gb[uiAxisNo].Diag,
        Axis               := Axis);
      (* check next axis *)
      uiAxisNo := uiAxisNo + 1;
      (* proceed with STATE_DO -> check next configured axis *)
      uiState := STATE_CHK_AXIS;

    END_IF

  STATE_ERROR:
        Active  := FALSE;
        Error   := TRUE;
        IF( (Execute = FALSE) AND (bOldExecute = TRUE) ) THEN
          uiState := STATE_DO_NOTHING;
        END_IF
				
	ELSE
	  ErrorID    := STATE_MACHINE_ERROR;
		ErrorIdent.Table := USER1_TABLE;
		ErrorIdent.Additional1 := uiState;
    ErrorIdent.Additional2 := 0;
		uiState    := STATE_ERROR;  
END_CASE

(* Edge detection *)
bOldExecute := Execute;

END_FUNCTION_BLOCK

// IndraMotionMlc1/Application/AxisInterface/TE_AxisInterface
// Online changes in declaration of axis-interface need too much time -> not allowed because risk of F5180006 
// InhibitOnlineChange = 0x1000000 has to be set decimal 16777216
{attribute 'signature_flag' := '16777216'} 
FUNCTION_BLOCK TE_AxisInterface EXTENDS MB_AxisInterfaceType01
(*#############################################################################################
  #############################################################################################  

  General Header   
  ---------------------------------------------------------------------------------------------  
  Shortdescription       : AxisInterface Example 
  Version                : see Version Function
  Name                   : DCC/EAM (DT/KG)
  Date                   : see Version Function
  Company                : see Version Function
  Target                 : see Version Function
  Functional description : Location in order to extend the AxisInterface functionality
  Handling specials      : This functionality is automatically assigned to the task the approriate
                           axis is assigned to
  ---------------------------------------------------------------------------------------------  
  
  Additional Header   
  ---------------------------------------------------------------------------------------------  

  ---------------------------------------------------------------------------------------------  

###############################################################################################  
###############################################################################################*)
(*
                                     ******************
                                     *   DISCLAIMER   *
                                     ******************
   It is acknowledged that with regard to these software programs and program modules free of
   charge, Bosch Rexroth's usually practised, in-house test and release procedures have not 
   been accomplished. These software programs and program modules free of charge serve only as
   an example for possible applications.  They are intended as a help in order to obtain addi-
   tional experience regarding function, operation, performance and capacity of a maybe later 
   issued series release. Therefore Bosch Rexroth disclaims any liability and rejects to assume
   responsibility that these software programs or program modules, including any information 
   and data stored in those programs, are suitable for any intended use or that these programs
   will work without errors in any combination with the data processing environment. Providing
   you with these software programs shall neither constitute a claim for technical support nor
   for any other remedy for defects. Any claims for damages of any nature and for any legal
   reason arising from installing or using these software programs or program modules are ex-
   cluded, unless these damages was caused by Bosch Rexroth`s statutory representatives or em-
   ployees by wilful misconduct or by gross negligence or liability is compulsory in accordance
   with the German product liability law. In any case Bosch Rexroth`s liability for any conse-
   quential or incidental damages such as, but not limited to loss of profit, loss of pro-
   duction or loss of data is excluded.      
*)
(*---------------------------------------------------------------------------------------------*)

VAR_INPUT
	// Internal references to the extension
    // this references include the base and the extensions, the refererences without Ext include only the base 
    (* arAxisCtrl_gb *)
	{attribute 'no_copy'}
    AdminCtrlExt     : REFERENCE TO TE_AXIS_ADMINISTRATION; (* Administration of the axis *)
	{attribute 'no_copy'}
    PosModeCtrlExt   : REFERENCE TO TE_AXIS_POSITIONING;    (* Operating mode absolute positioning *)
	{attribute 'no_copy'}
    VelModeCtrlExt   : REFERENCE TO TE_AXIS_VELOCITY;       (* Operating mode velocity control *)
	{attribute 'no_copy'}
    SyncModeCtrlExt  : REFERENCE TO TE_AXIS_SYNCHRONISATION;(* Operating mode synchronisation (phs,vel,and cam)*)
	{attribute 'no_copy'}
    TorqueModeCtrlExt: REFERENCE TO TE_AXIS_TORQUE;       (* Operating mode torque-/force control*)	
    (* arAxisStatus_gb *)
	{attribute 'no_copy'}
    AdminStatusExt   : REFERENCE TO TE_AXIS_ADMIN_STATUS;   (* Status administration of the axis *)
	{attribute 'no_copy'}
    DiagStatusExt    : REFERENCE TO TE_AXIS_DIAGNOSIS;      (* Axis diagnosis information, error, warning.... *)
	{attribute 'no_copy'}
    PosStatusExt     : REFERENCE TO TE_AXIS_POS_STATUS;     (* Status operating mode positioning *)
	{attribute 'no_copy'}
    VelStatusExt     : REFERENCE TO TE_AXIS_VEL_STATUS;     (* Status operating mode velocity control *)
	{attribute 'no_copy'}
    SyncModeStatusExt: REFERENCE TO TE_AXIS_SYNC_STATUS;    (* Status op mode synchronisation (phs,vel,and cam)*)
    // add user extensions below here
	{attribute 'no_copy'}
    SetupMode: REFERENCE TO TE_AXIS_SETUP_MODE;
	{attribute 'no_copy'} 
    SetupModeAck: REFERENCE TO TE_AXIS_SETUP_MODE_STATUS;
	{attribute 'no_copy'} 
	  AxisData_HMI: REFERENCE TO TE_AXIS_DATA_STATUS;
END_VAR
VAR_OUTPUT

END_VAR
VAR
  udiCycleCntInP4: UDINT; // count cycles in P4 to spread the parameter write load
  //######  SetupMode ######## 
  bLatchSetupModeEnable:  BOOL;
  enOriAxisMode:  MB_AXIS_MODE; 	// stored OpMode, when SetupMode is activated. reset when SetupMode is left
  enMyActAxisMode:  MB_AXIS_MODE;	// actual Setup-OpMode, used to detect when the OpMode is changed during active SetupMode  
  uiHomingState: UINT;
  // define as RETAIN (global) when arAxisCtrl_gb is RETAIN 
  bOriValuesStored:  BOOL;
  rOriVel:  REAL;
  rOriAccel:  REAL;
  rOriDecel:  REAL;
  rOriDistance: REAL;
  rOriVelPos: REAL;
  rOriAccelPos: REAL;
  rOriDecelPos: REAL;
  rSetupModePosDiff: REAL;   // difference for jogging in positioning mode

  //######  Homing ########
  bHomingOld: BOOL:=FALSE;  // to detect the falling edge
  bHomingRemovedBeforeFinished: BOOL:= FALSE;
  bAbsoluteEncoder: BOOL:=FALSE;
  diParameterS277: DINT:=0;
  MB_ReadParameterS277: MB_ReadParameter;

  //######  AngleOffset ######## 
  // Remember AngleOffset to write only on changes 
  rLastAngleOffset:  REAL; 
  // Write AngleOffset 
  fbWrAngleOffs:       MB_WriteRealParameter;
  bExecWrAngleOffs:    BOOL:=FALSE;
  bRestartAngleOffs:   BOOL:=TRUE;  // restart when entering sync op-mode

  //######  SyncAcceleration ######## 
  // Remember SyncAcceleration to write only on changes 
  rLastSyncAcc:      REAL; 
  // Write SyncAcceleration 
  fbWrSyncAcc:       MB_WriteRealParameter;
  bExecWrSyncAcc:    BOOL:=FALSE;
  bRestartSyncAcc:   BOOL:=TRUE;  // restart when entering sync op-mode

  //######  Syncvelocity ######## 
  // Remember Syncvelocity to write only on changes 
  rLastSyncVel:      REAL; 
  // Write SyncAcceleration 
  fbWrSyncVel:       MB_WriteRealParameter;
  bExecWrSyncVel:    BOOL:=FALSE;
  bRestartSyncVel:   BOOL:=TRUE;  // restart when entering sync op-mode
  
  //######  PhasingMaster ######## 
  fbAxisPhasing: MB_Phasing;
  bExecPhasing:    BOOL:=FALSE;
  rOldPhaseShift:  REAL;        // change detection
  bRestartPhasing: BOOL:=TRUE;  // restart when entering sync op-mode
  
  //######  RetriggerOpMode ######## 
  bRetriggerOpModeOld: BOOL;
  bOriginalOpMode: MB_AXIS_MODE;
  bOpModeChanged: BOOL;
	
	//######  Activate PM for special axis errors ########
  bOriginalPM: BOOL;
	uiStatePM: UINT :=STATE_ERR_IDLE;
  
END_VAR
VAR CONSTANT  
  STATE_HOMING_START         :UINT := 0;
  STATE_HOMING_READ_S277     :UINT := 1;
  STATE_HOMING_ABS_REAL_AXIS :UINT := 2;
  STATE_HOMING_INC_REAL_AXIS :UINT := 3;
  STATE_HOMING_VIRT_AXIS     :UINT := 5;
  STATE_HOMING_FINISHED      :UINT := 6;
  STATE_HOMING_NOT_POSSIBLE  :UINT := 9;
  STATE_HOMING_NOT_IMPLEMENT :UINT := 10;
  STATE_HOMING_ERROR         :UINT := 11;

  // States of special error handling  
	STATE_ERR_IDLE             :UINT := 0;
	STATE_ERR_ACTIVATE_PM      :UINT := 1;
	STATE_ERR_ACTIVATE_OM      :UINT := 2;

  // state machine error
  HOMING_STATE_MACHINE_ERR: ERROR_STRUCT := ( Table := USER10_TABLE, Additional1 := 16#00004201, Additional2 := 16#00000000);
  // Homing not implemented for control axis
  HOMING_CONFIGURATION_ERR: ERROR_STRUCT := ( Table := USER10_TABLE, Additional1 := 16#00004202, Additional2 := 16#00000000);
  // SetupMode is only allowed when in Modeab or ModeAH
  SETUPMODE_OPMODE_ERR: ERROR_STRUCT := ( Table := USER10_TABLE, Additional1 := 16#00004203, Additional2 := 16#00000000);
  
  rFACTOR_VEL_TO_POS:    REAL:= 0.25; // factor for calculating distance when jogging in positioning mode
  rSETUP_MODE_POS_DIFF2: REAL:= 0.1;  // 2nd difference for jogging in positioning mode (relative positioning)
END_VAR

// Handle RetriggerOpMode 
// Do this before calling the base FB to be able to overwrite the OpMode set cyclic by the user.
actRetriggerOpMode();
// Activate PM for special axis errors. In case of drive error F8022 and F8042 switch to PM to clear this error.
// Do this before calling the base FB to be able to overwrite the paramLevel set cyclic by the user.  
//actPMSpecialErrors(); // Comment out this line in case this reaction is not required. This saves execution time.

(* call the base FB, call it first, to have the information AdminStatus.Active actual *)
SUPER^();

(* 2nd check, if the axis is active *)
IF AdminStatus.Active = FALSE THEN	
  RETURN;
END_IF;
// Check if we are in bb. A-0-0021 is read internal by the MB_AxisInterfaceType01
// Bit 12 of A-0-0021 means "Axis is in operation mode (P4)" 
// When all axes in parallel write parameters, we overload the system. So we
// count the cycles and distribute the load with using the axis address  
IF AxisData[AdminCtrl.Axis.AxisNo].Axis_OperationMode = TRUE THEN 
  udiCycleCntInP4 := udiCycleCntInP4 + 1;
ELSE
  udiCycleCntInP4 := 0;
END_IF

(* add your extensions below here, keep the elements above
   Erweiterungen hier einfuegen, Elemente oberhalb nicht veraendern *)
(* user extensions | Anwender Erweiterungen *)

(* Jog/Home an axis within the AxisInterface *)
actSetupMode();

(* Write the Angle offset begin of profile A-0-2730 *)
actAngleOffset();

(* Write the Sync Acceleration into A-0-2791 *)
(* and the Sync Velocity into A-0-2790 *)
actSyncAccVel();

(* Handle PhasingMaster *)
actPhaseShift();

(* copy AxisData status informations to AxisData_HMI structure to transmit to HMI *)
actCopyAxisData_HMI();

ACTION actAngleOffset:
// Implements writing the angle offset into parameter A-0-2730
// Check if we are in bb. Otherwise we get errors.
// Do this only when sync is supported and the parameters are available
// AND not for IPO-Control. A-0-2730 is only needed for Cam.
// Distribute the load with using the axis address
IF AxisData[AdminCtrlExt.Axis.AxisNo].Axis_OperationMode = TRUE   AND
   AdminStatusExt.AxisFeatures.OPMODE_SYNC = TRUE                 AND 
   NOT AdminStatusExt.AxisFeatures.IPO_CONTROL                    AND
   (udiCycleCntInP4 > DINT_TO_UDINT(2 * AdminCtrlExt.Axis.AxisNo))    THEN 
  // write angle offset when changed 
  IF SyncModeCtrlExt.AngleOffset <> rLastAngleOffset OR bRestartAngleOffs THEN
    // changed value OR 1st time in Operation-Mode
    IF bExecWrAngleOffs = TRUE THEN
      // transmission is active, we need a new edge. Abort the actual transmission.
      bExecWrAngleOffs := FALSE;
    ELSE
      // no transmission active or we aborted the transmission, generate a new rising edge 
      bExecWrAngleOffs := TRUE;
      // remember old value 
      rLastAngleOffset := SyncModeCtrlExt.AngleOffset;
      bRestartAngleOffs := FALSE;
		END_IF
    // start transmission 
    SyncModeStatusExt.AngleOffsetDone := FALSE;
  END_IF
  IF fbWrAngleOffs.Done = TRUE THEN 
    // finished GOOD transmission 
    SyncModeStatusExt.AngleOffsetDone := TRUE;
    bExecWrAngleOffs := FALSE;
  ELSIF fbWrAngleOffs.Error = TRUE THEN  
    // finished BAD transmission 
    bExecWrAngleOffs := FALSE;
    SUPER^.mSetError( Error      := TRUE, 
                      ErrorID    := fbWrAngleOffs.ErrorID, 
                      ErrorIdent := fbWrAngleOffs.ErrorIdent);
  END_IF  
  // for IPO-Drive -> call write parameter FB 
  fbWrAngleOffs(
	Execute:= bExecWrAngleOffs, 
	ParameterNumber:= FP_A_0_2730, 
	Value:= SyncModeCtrlExt.AngleOffset, 
	Axis:= AdminCtrlExt.Axis );	
ELSE
  // reset FBs when not in bb 
  fbWrAngleOffs( Execute:= FALSE, Axis:= AdminCtrlExt.Axis );	
END_IF	
// to avoid service channel transmissions (interFIation drive), place the P-0-0061 into 
// an MDT data container (here e.g. container A) and write to the data container
//AxisData[AdminCtrlExt.Axis].dwUserCmdDataA_q.REAL_ := SyncModeCtrlExt.AngleOffset;
END_ACTION

ACTION actCopyAxisData_HMI:
// copy AxisData status informations to AxisData_HMI structure to transmit to HMI

AxisData_HMI.dwMotionProfileStatusBits_i    	:=	AxisData[AdminCtrlExt.Axis.AxisNo].dwMotionProfileStatusBits_i;	
AxisData_HMI.FlexProfil_Sync                    :=  AxisData[AdminCtrlExt.Axis.AxisNo].FlexProfil_Sync;                 
AxisData_HMI.FlexProfil_Active                  :=  AxisData[AdminCtrlExt.Axis.AxisNo].FlexProfil_Active;               
AxisData_HMI.FlexProfil_WaitForSwitching        :=  AxisData[AdminCtrlExt.Axis.AxisNo].FlexProfil_WaitForSwitching;     
AxisData_HMI.FlexProfil_Set0_Checked            :=  AxisData[AdminCtrlExt.Axis.AxisNo].FlexProfil_Set0_Checked;         
AxisData_HMI.FlexProfil_Set0_Ok                 :=  AxisData[AdminCtrlExt.Axis.AxisNo].FlexProfil_Set0_Ok;              
AxisData_HMI.FlexProfil_Set1_Checked            :=  AxisData[AdminCtrlExt.Axis.AxisNo].FlexProfil_Set1_Checked;         
AxisData_HMI.FlexProfil_Set1_Ok                 :=  AxisData[AdminCtrlExt.Axis.AxisNo].FlexProfil_Set1_Ok;              
AxisData_HMI.FlexProfil_Set2_Checked            :=  AxisData[AdminCtrlExt.Axis.AxisNo].FlexProfil_Set2_Checked;         
AxisData_HMI.FlexProfil_Set2_Ok                 :=  AxisData[AdminCtrlExt.Axis.AxisNo].FlexProfil_Set2_Ok;              
AxisData_HMI.FlexProfil_Set3_Checked            :=  AxisData[AdminCtrlExt.Axis.AxisNo].FlexProfil_Set3_Checked;         
AxisData_HMI.FlexProfil_Set3_Ok                 :=  AxisData[AdminCtrlExt.Axis.AxisNo].FlexProfil_Set3_Ok;              
AxisData_HMI.FlexProfil_EvtSet0_Checked         :=  AxisData[AdminCtrlExt.Axis.AxisNo].FlexProfil_EvtSet0_Checked;      
AxisData_HMI.FlexProfil_EvtSet0_Ok              :=  AxisData[AdminCtrlExt.Axis.AxisNo].FlexProfil_EvtSet0_Ok;           
AxisData_HMI.FlexProfil_EvtSet1_Checked         :=  AxisData[AdminCtrlExt.Axis.AxisNo].FlexProfil_EvtSet1_Checked;      
AxisData_HMI.FlexProfil_EvtSet1_Ok              :=  AxisData[AdminCtrlExt.Axis.AxisNo].FlexProfil_EvtSet1_Ok;           
AxisData_HMI.FlexProfil_EvtSet2_Checked         :=  AxisData[AdminCtrlExt.Axis.AxisNo].FlexProfil_EvtSet2_Checked;      
AxisData_HMI.FlexProfil_EvtSet2_Ok              :=  AxisData[AdminCtrlExt.Axis.AxisNo].FlexProfil_EvtSet2_Ok;           
AxisData_HMI.FlexProfil_EvtSet3_Checked         :=  AxisData[AdminCtrlExt.Axis.AxisNo].FlexProfil_EvtSet3_Checked;      
AxisData_HMI.FlexProfil_EvtSet3_Ok              :=  AxisData[AdminCtrlExt.Axis.AxisNo].FlexProfil_EvtSet3_Ok;           
AxisData_HMI.dwFlexProfileEventStatusBits_i     :=  AxisData[AdminCtrlExt.Axis.AxisNo].dwFlexProfileEventStatusBits_i; 
AxisData_HMI.Axis_CamTab_0                      :=  AxisData[AdminCtrlExt.Axis.AxisNo].Axis_CamTab_0;                   
AxisData_HMI.Axis_CamTab_1                      :=  AxisData[AdminCtrlExt.Axis.AxisNo].Axis_CamTab_1;                   
AxisData_HMI.Axis_CamTab_2                      :=  AxisData[AdminCtrlExt.Axis.AxisNo].Axis_CamTab_2;                   
AxisData_HMI.Axis_CamSwitching                  :=  AxisData[AdminCtrlExt.Axis.AxisNo].Axis_CamSwitching;               
AxisData_HMI.Axis_InVelocity                    :=  AxisData[AdminCtrlExt.Axis.AxisNo].Axis_InVelocity;                 
AxisData_HMI.Axis_Standstill                    :=  AxisData[AdminCtrlExt.Axis.AxisNo].Axis_Standstill;                 
AxisData_HMI.Axis_InPosition                    :=  AxisData[AdminCtrlExt.Axis.AxisNo].Axis_InPosition;      
AxisData_HMI.Axis_InSynchron                    :=  AxisData[AdminCtrlExt.Axis.AxisNo].Axis_InSynchron;                 
AxisData_HMI.Axis_Warning                       :=  AxisData[AdminCtrlExt.Axis.AxisNo].Axis_Warning;                    
AxisData_HMI.Axis_Error                         :=  AxisData[AdminCtrlExt.Axis.AxisNo].Axis_Error;                      
AxisData_HMI.Axis_Homed                         :=  AxisData[AdminCtrlExt.Axis.AxisNo].Axis_Homed;                      
AxisData_HMI.Axis_InTorque                      :=  AxisData[AdminCtrlExt.Axis.AxisNo].Axis_InTorque;                   
AxisData_HMI.Axis_OperationMode                 :=  AxisData[AdminCtrlExt.Axis.AxisNo].Axis_OperationMode;              
AxisData_HMI.Axis_Inbb                          :=  AxisData[AdminCtrlExt.Axis.AxisNo].Axis_Inbb;                       
AxisData_HMI.Axis_InAb                          :=  AxisData[AdminCtrlExt.Axis.AxisNo].Axis_InAb;                       
AxisData_HMI.Axis_Power                         :=  AxisData[AdminCtrlExt.Axis.AxisNo].Axis_Power;                      
AxisData_HMI.Axis_CmdActive                     :=  AxisData[AdminCtrlExt.Axis.AxisNo].Axis_CmdActive;                  
AxisData_HMI.Axis_ErrInProgress                 :=  AxisData[AdminCtrlExt.Axis.AxisNo].Axis_ErrInProgress;              
AxisData_HMI.Axis_CyclicPosChannelOpen          :=  AxisData[AdminCtrlExt.Axis.AxisNo].Axis_CyclicPosChannelOpen;       
AxisData_HMI.Axis_InMasterPhaseOffset           :=  AxisData[AdminCtrlExt.Axis.AxisNo].Axis_InMasterPhaseOffset;        
AxisData_HMI.Axis_CyclicTrqChannelOpen          :=  AxisData[AdminCtrlExt.Axis.AxisNo].Axis_CyclicTrqChannelOpen;       
AxisData_HMI.Axis_CyclicVelChannelOpen          :=  AxisData[AdminCtrlExt.Axis.AxisNo].Axis_CyclicVelChannelOpen;       
AxisData_HMI.Axis_CyclicAnaChannelOpen          :=  AxisData[AdminCtrlExt.Axis.AxisNo].Axis_CyclicAnaChannelOpen;       
AxisData_HMI.ErrorStop                          :=  AxisData[AdminCtrlExt.Axis.AxisNo].ErrorStop;                       
AxisData_HMI.Stopping                           :=  AxisData[AdminCtrlExt.Axis.AxisNo].Stopping;                        
AxisData_HMI.Homing                             :=  AxisData[AdminCtrlExt.Axis.AxisNo].Homing;                          
AxisData_HMI.PowerOn                            :=  AxisData[AdminCtrlExt.Axis.AxisNo].PowerOn;                         
AxisData_HMI.DiscreteMotion                     :=  AxisData[AdminCtrlExt.Axis.AxisNo].DiscreteMotion;                  
AxisData_HMI.ContinuousMotion                   :=  AxisData[AdminCtrlExt.Axis.AxisNo].ContinuousMotion;                
AxisData_HMI.SynchronizedMotion                 :=  AxisData[AdminCtrlExt.Axis.AxisNo].SynchronizedMotion;              
AxisData_HMI.Standstill                         :=  AxisData[AdminCtrlExt.Axis.AxisNo].Standstill;                      
AxisData_HMI.CoordinatedMotion                  :=  AxisData[AdminCtrlExt.Axis.AxisNo].CoordinatedMotion;               
AxisData_HMI.ControlledMotion                   :=  AxisData[AdminCtrlExt.Axis.AxisNo].ControlledMotion;                
AxisData_HMI.dwAxisCondition_i                  :=  AxisData[AdminCtrlExt.Axis.AxisNo].dwAxisCondition_i;               
AxisData_HMI.rActualPosition_i                  :=  AxisData[AdminCtrlExt.Axis.AxisNo].rActualPosition_i;               
AxisData_HMI.rActualVelocity_i                  :=  AxisData[AdminCtrlExt.Axis.AxisNo].rActualVelocity_i;               
AxisData_HMI.rActualTorqueForce_i               :=  AxisData[AdminCtrlExt.Axis.AxisNo].rActualTorqueForce_i;            
AxisData_HMI.wUserActualDataBitA_i              :=  AxisData[AdminCtrlExt.Axis.AxisNo].wUserActualDataBitA_i;          
AxisData_HMI.wUserActualDataBitB_i              :=  AxisData[AdminCtrlExt.Axis.AxisNo].wUserActualDataBitB_i;          
AxisData_HMI.wUserActualDataBitC_i              :=  AxisData[AdminCtrlExt.Axis.AxisNo].wUserActualDataBitC_i;          
AxisData_HMI.wUserActualDataBitD_i              :=  AxisData[AdminCtrlExt.Axis.AxisNo].wUserActualDataBitD_i;          
AxisData_HMI.dwUserActualDataA_i                :=  AxisData[AdminCtrlExt.Axis.AxisNo].dwUserActualDataA_i;             
AxisData_HMI.dwUserActualDataB_i                :=  AxisData[AdminCtrlExt.Axis.AxisNo].dwUserActualDataB_i;             
AxisData_HMI.dwUserActualDataC_i                :=  AxisData[AdminCtrlExt.Axis.AxisNo].dwUserActualDataC_i;             
AxisData_HMI.dwUserActualDataD_i                :=  AxisData[AdminCtrlExt.Axis.AxisNo].dwUserActualDataD_i;             
AxisData_HMI.dwUserActualDataE_i                :=  AxisData[AdminCtrlExt.Axis.AxisNo].dwUserActualDataE_i;             
AxisData_HMI.dwUserActualDataF_i                :=  AxisData[AdminCtrlExt.Axis.AxisNo].dwUserActualDataF_i;
END_ACTION

ACTION actPhaseShift:
//***************************************************************
// Implements a PhasingMaster with the function block MB_Phasing
//***************************************************************
//********* handle phase offset when sync-mode is active *******
IF( ((ANY_TO_DWORD(AdminStatusExt._OpModeAck) AND Global_AxIf_Const.MASK_MODE_PHASE_SHIFT) <> 0) )THEN
  IF( rOldPhaseShift <> SyncModeCtrlExt.PhaseShift) OR bRestartPhasing THEN
    // changed value OR 1st time in Sync-Mode
    IF bExecPhasing = TRUE THEN
      // transmission is active, we need a new edge. Abort the actual transmission.
      bExecPhasing := FALSE;
    ELSE
      // no transmission active or we aborted the transmission, generate a new rising edge 
      bExecPhasing := TRUE;
      // remember old value 
      rOldPhaseShift := SyncModeCtrlExt.PhaseShift;
      bRestartPhasing := FALSE;
		END_IF
    // start transmission 
	  SyncModeStatusExt.PhasingMasterDone := FALSE;
  END_IF
  IF fbAxisPhasing.Done THEN
    // finished GOOD transmission 
		SyncModeStatusExt.PhasingMasterDone := TRUE;
		bExecPhasing := FALSE;
  ELSIF (fbAxisPhasing.Error = TRUE) THEN
    // finished BAD transmission 
		bExecPhasing := FALSE;
    SUPER^.mSetError( Error      := TRUE, 
                      ErrorID    := fbAxisPhasing.ErrorID, 
                      ErrorIdent := fbAxisPhasing.ErrorIdent);
  END_IF
ELSE
  SyncModeStatusExt.PhasingMasterDone := FALSE; // Reset, when no Sync-Mode active 
	// Reset, when no sync-mode is active
	bExecPhasing := FALSE;
  // Start a new transmission so PhasingMasterDone is set again after a re-start
  bRestartPhasing := TRUE;
END_IF // end of 'IF( (INT_TO_WORD(AdminStatusExt._OpMode.enAck) AND MASK_MODE_PHASE_OFFSET) <> 0 ) THEN'
// keep the FB always up-to-date 
fbAxisPhasing(
	Execute      := bExecPhasing,
	PhaseShift   := SyncModeCtrlExt.PhaseShift,
	Velocity     := SyncModeCtrlExt.PhaseShiftVel,
	Acceleration := SyncModeCtrlExt.PhaseShiftAcc,
	Axis         := AdminCtrlExt.Axis );
END_ACTION

ACTION actPMSpecialErrors:
// Activate PM of the axis if special drive errors occur 

{IF defined(variable: AdminCtrl.ParamLevel)}
CASE uiStatePM OF
  
STATE_ERR_IDLE: 
  // ---------------------------------------------------------
  // Idle state --> do nothing
	// ---------------------------------------------------------
  // Wait until F8022 or F8042 error occurs   
	IF (DiagStatusExt.Error = TRUE) AND((DiagStatus.Number = 16#F2008022) OR (DiagStatus.Number = 16#F2008042)) THEN
		bOriginalPM := AdminCtrl.ParamLevel;
    uiStatePM := STATE_ERR_ACTIVATE_PM;	
	END_IF
	
STATE_ERR_ACTIVATE_PM:
  // ---------------------------------------------------------
  // Command axis to Parameter mode "PM"  
	// ---------------------------------------------------------
  AdminCtrl.ParamLevel := TRUE;
 
	// Wait until error disappears
	IF (DiagStatusExt.Error = FALSE ) THEN
    uiStatePM := STATE_ERR_ACTIVATE_OM;	
	END_IF
 
STATE_ERR_ACTIVATE_OM: 
  // ---------------------------------------------------------
  // Command axis to Operation Mode "OM" 
  // --------------------------------------------------------- 
  AdminCtrl.ParamLevel := FALSE;
 
  // Wait untill axis is in OM 
  IF AxisData[AdminCtrl.Axis.AxisNo].Axis_OperationMode = TRUE THEN
    uiStatePM := STATE_ERR_IDLE;	
		AdminCtrl.ParamLevel := bOriginalPM;
	END_IF

END_CASE
{END_IF}
;
END_ACTION

ACTION actRetriggerOpMode:
// Restart the same OpMode again, e.g. MoveRelative with same distance
// Detect rising edge on input RetriggerOpMode
IF AdminCtrlExt.RetriggerOpMode AND NOT bRetriggerOpModeOld THEN
  // set ModeExternalFb for one cycle
    bOriginalOpMode := AdminCtrlExt._OpMode.en ;
    AdminCtrlExt._OpMode.en := ModeExternalFb;
    bOpModeChanged :=TRUE;
ELSIF bOpModeChanged THEN
    // reset OpMode to original in next cycle
    AdminCtrl._OpMode.en := bOriginalOpMode;
    bOpModeChanged :=FALSE; 
END_IF
bRetriggerOpModeOld  := AdminCtrlExt.RetriggerOpMode;
END_ACTION

ACTION actSetupMode:
//***************************************************************
// Implements a jogging based on velocity mode
// Implements homing depending on the axis type
//   Virtual axis: move absolute to 360 degrees
//   Real axis: depending on parameter S-0-0277 ModeHoming or SetAbsRef
//***************************************************************
// Do nothing, when not enabled... 
IF SetupMode.Enable = TRUE THEN
  // Positive edge of Enable ?
  IF NOT bLatchSetupModeEnable THEN
		// SetupMode is only allowed when in ModeAb or ModeAH 
		IF( (AdminCtrlExt._OpMode.en=ModeAH) OR (AdminCtrlExt._OpMode.en=ModeAb) ) THEN
      // store original values 
      rOriVel          := VelModeCtrlExt.Velocity;
      rOriAccel        := VelModeCtrlExt.Acceleration;
      rOriDecel        := AdminCtrlExt.StopDeceleration;  // Defdb00116851 / Defdb00116875  
      rOriDistance     := PosModeCtrlExt.Distance;
      rOriVelPos       := PosModeCtrlExt.Velocity;
      rOriAccelPos     := PosModeCtrlExt.Acceleration;
      rOriDecelPos     := PosModeCtrlExt.Deceleration;
      enOriAxisMode    := AdminCtrlExt._OpMode.en;
  	  bOriValuesStored := TRUE;
      // activate mode AH
      AdminCtrlExt._OpMode.en := ModeAH;
  	  enMyActAxisMode 	      := ModeAH;
  	  uiHomingState 	      := STATE_HOMING_START;
  	  //SetupModeAck.EnableAck  := TRUE; // Acknowledge SetupMode
    ELSE
      // actual not allowed to activate SetupMode
      SUPER^.mSetError( Error      := TRUE, 
                        ErrorID    := RESOURCE_ERROR, 
             	        ErrorIdent := SETUPMODE_OPMODE_ERR);
  	  bOriValuesStored:= FALSE;
    END_IF  
  END_IF // IF NOT bLatchSetupModeEnable THEN
  
  // Check if someone did overwrite our OpMode command?
  IF( (AdminCtrlExt._OpMode.en <> enMyActAxisMode) AND (SetupModeAck.EnableAck = TRUE) ) THEN
    SetupModeAck.EnableAck := FALSE; // remove acknowledge SetupMode
	
  ELSIF SetupMode.Enable = TRUE THEN
  
    IF SetupMode.JogPosControl = FALSE THEN
    //***************************************************************
      // Jogging in velocity mode
    //***************************************************************
    // Jog positive direction 
    IF SetupMode.JogPlus AND NOT SetupMode.JogMinus THEN
      VelModeCtrlExt.Acceleration	:= SetupMode.Accel;
      AdminCtrlExt.StopDeceleration	:= SetupMode.Accel;  // Defdb00116851 / Defdb00116875
      VelModeCtrlExt.Velocity := SetupMode.Vel;
	  AdminCtrlExt._OpMode.en := ModeVel; 
      enMyActAxisMode := ModeVel; 
    	// Jog negative direction 
    ELSIF SetupMode.JogMinus AND NOT SetupMode.JogPlus THEN
      VelModeCtrlExt.Acceleration	:= SetupMode.Accel;
      AdminCtrlExt.StopDeceleration	:= SetupMode.Accel;  // Defdb00116851 / Defdb00116875
      VelModeCtrlExt.Velocity := -SetupMode.Vel;
  	AdminCtrlExt._OpMode.en := ModeVel;  
  	enMyActAxisMode         := ModeVel;
    ELSIF AdminCtrlExt._OpMode.en = ModeVel THEN
      // switch back when coming from Jog (do not disturb homing)
  	AdminCtrlExt._OpMode.en := ModeAH;
  	enMyActAxisMode         := ModeAH;
    END_IF
    ELSE
      //*************************************************************************************
      // Jogging in relative positioning control, position control loop monitoring is active. 
      // Position limit value monitoring is active, when the axis is referenced.
      //*************************************************************************************
      rSetupModePosDiff := SetupMode.Vel * rFACTOR_VEL_TO_POS; // use a larger distance with higher speed
      // Jog positive direction 
      IF SetupMode.JogPlus AND NOT SetupMode.JogMinus THEN
        PosModeCtrlExt.Acceleration	:= SetupMode.Accel;
        PosModeCtrlExt.Deceleration	:= SetupMode.Accel;
        AdminCtrlExt.StopDeceleration	:= SetupMode.Accel; 
        PosModeCtrlExt.Velocity := SetupMode.Vel;
        // use relative positioning for jogging
        // + -> toggle between two distances to generate a continuous movement
        IF rSetupModePosDiff = PosModeCtrlExt.Distance THEN
          PosModeCtrlExt.Distance := rSetupModePosDiff+rSETUP_MODE_POS_DIFF2;
        ELSE
          PosModeCtrlExt.Distance := rSetupModePosDiff;
        END_IF  
        AdminCtrlExt._OpMode.en := ModePosRel;
        enMyActAxisMode := ModePosRel; 
        // Jog negative direction 
      ELSIF SetupMode.JogMinus AND NOT SetupMode.JogPlus THEN
        PosModeCtrlExt.Acceleration	:= SetupMode.Accel;
        PosModeCtrlExt.Deceleration	:= SetupMode.Accel;
        AdminCtrlExt.StopDeceleration	:= SetupMode.Accel;
        PosModeCtrlExt.Velocity := SetupMode.Vel;
        // use relative positioning for jogging
        // - -> toggle between two negative distances to generate a continuous movement
        IF -rSetupModePosDiff = PosModeCtrlExt.Distance THEN
          PosModeCtrlExt.Distance := -(rSetupModePosDiff+rSETUP_MODE_POS_DIFF2);
        ELSE
          PosModeCtrlExt.Distance := -rSetupModePosDiff;
        END_IF  
        AdminCtrlExt._OpMode.en := ModePosRel; 
        enMyActAxisMode := ModePosRel; 
      // switch off 
      ELSIF AdminCtrlExt._OpMode.en = ModePosRel THEN
        // switch back when coming from Jog (do not disturb homing)
        AdminCtrlExt._OpMode.en := ModeAH;
        enMyActAxisMode         := ModeAH;
      END_IF
		END_IF // end of 'IF SetupMode.JogPosControl = FALSE THEN'

    //***************************************************************
    // Implements homing depending on the axis type
    // Virtual axis: move absolute to 360 degrees
    // Real axis with closed loop: depending on parameter S-0-0277 ModeHoming or SetAbsRef
    // Controller axis: not implemented, change to real axis when S-0-0277/S-0-0477 available 
    //***************************************************************
  (* Parameter S277 Bit7/6: only read)
				
		7/6	absolute encoder
		x0: absolute encoder not possible (Bit 7 not in use)
		01: absolute encoder is active)
		11: absolute encoder is possible but deactivated *)

    CASE uiHomingState OF
  
    STATE_HOMING_START:		
        // #####################################################################  
      	IF( (AdminStatusExt.AxisFeatures.OPMODE_POS = FALSE) OR
            ((DV_Axis[AdminCtrlExt.Axis.AxisNo].A_0_0024 AND A24_CMD_DECOUPLED_MASK) = A24_BIT_CMD_DECOUPLED) 
          ) THEN   
          uiHomingState := STATE_HOMING_NOT_POSSIBLE; // can not be homed, e.g. open loop
        ELSIF (AdminStatusExt.AxisFeatures.CONTROLLER_AXIS = TRUE) THEN // when S-0-0277/S-0-0447 are not available  
          uiHomingState := STATE_HOMING_NOT_IMPLEMENT; // controller axis without S-0-0277/S-0-0447          
        ELSIF AdminStatusExt.AxisFeatures.REAL_AXIS = TRUE 
          (* OR (AdminStatusExt.AxisFeatures.CONTROLLER_AXIS = TRUE) // when S-0-0277/S-0-0447 available *) THEN
					uiHomingState := STATE_HOMING_READ_S277;   // continue with read S-0-0277
      	ELSIF AdminStatusExt.AxisFeatures.VIRTUAL_AXIS = TRUE THEN
					uiHomingState := STATE_HOMING_VIRT_AXIS;   // continue with homing virtual axis
      	ELSE 
      	  // undefined axis type
   	  	  SUPER^.mSetError( Error      := TRUE, 
       		                  ErrorID    := RESOURCE_ERROR, 
           		              ErrorIdent := HOMING_CONFIGURATION_ERR);
   	  	  uiHomingState := STATE_HOMING_ERROR;   // continue with error
  		  END_IF
  
    STATE_HOMING_READ_S277:
        // #####################################################################  
      	// first read S-0-0277 when SetupMode is activated
	 			MB_ReadParameterS277(
    		Enable:= TRUE, 
    		ParameterNumber:= FP_S_0_0277, 
    		Axis:= AdminCtrlExt.Axis );
   		  IF MB_ReadParameterS277.Done = TRUE THEN
					// store Value   
					diParameterS277 := MB_ReadParameterS277.Value;
					IF 	(diParameterS277.6 AND NOT diParameterS277.7) OR diParameterS277.8 THEN
		    	  // absolute encoder
						bAbsoluteEncoder := TRUE;
        	  uiHomingState := STATE_HOMING_ABS_REAL_AXIS; // continue with homing an absolute real axis
					ELSE
		    	  // incremental encoder
						bAbsoluteEncoder := FALSE;
        	  uiHomingState := STATE_HOMING_INC_REAL_AXIS; // continue with homing an incremental real axis
					END_IF
					// RESET FB  
    		MB_ReadParameterS277(
       		Enable:= FALSE, 
      		ParameterNumber:= FP_S_0_0277, 
      		Axis:= AdminCtrlExt.Axis );
      	ELSIF MB_ReadParameterS277.Error = TRUE THEN
    		  SUPER^.mSetError( Error      := TRUE, 
                            ErrorID    := MB_ReadParameterS277.ErrorID, 
                            ErrorIdent := MB_ReadParameterS277.ErrorIdent);
					// RESET FB  
    		  MB_ReadParameterS277(
       		  Enable:= FALSE, 
      		  ParameterNumber:= FP_S_0_0277, 
      		  Axis:= AdminCtrlExt.Axis );
        	  uiHomingState := STATE_HOMING_ERROR;   // continue with error
  		  END_IF	// end of 'IF MB_ReadParameterS277.Done = TRUE THEN'		  
	
    STATE_HOMING_ABS_REAL_AXIS, STATE_HOMING_VIRT_AXIS:
        // ##################################################################### 
				SetupModeAck.EnableAck  := TRUE; // Acknowledge SetupMode 
    		// Homing for Real-Axis with absolute encoder
      	IF (SetupMode.Homing = TRUE) AND (bHomingOld = FALSE) THEN
       		// Set reference with absolute encoder
       		AdminCtrlExt._OpMode.en := ModeAB;
    			enMyActAxisMode         := ModeAB;
				// wait for Homing finished
      	ELSIF  AdminStatusExt.AbsRefCmdStatus = MB_SERCOS_DATA_END_OK THEN
					// command finished GOOD
					SetupModeAck.HomingAck := TRUE;
					uiHomingState := STATE_HOMING_FINISHED;
					IF SetupMode.Homing = FALSE THEN
		  		  // Input was removed. Switch back to ModeAH. HomingAck stays active for one cycle... 	
		  		  bHomingRemovedBeforeFinished := TRUE;	
					END_IF	
        // Note: problems with IndraDrive Cs. It takes time to switch to AB and the 
        // C0304 "command not allowed in AF" can happen so wait for PowerOff before 
        // setting the command set absolute reference
      	ELSIF (SetupMode.Homing = TRUE) AND 
              (AdminStatusExt._OpModeAck = ModeAb) THEN
       		AdminCtrlExt.SetAbsRef := TRUE;
				ELSIF ( (AdminStatusExt.AbsRefCmdStatus = MB_SERCOS_DATA_INTERRUPTED) OR	
	    	        (AdminStatusExt.AbsRefCmdStatus = MB_SERCOS_DATA_BREAK_ERROR) OR
								(AdminStatusExt.AbsRefCmdStatus = MB_SERCOS_DATA_DATUM_FAULT)    ) THEN
					// command finished BAD
					SetupModeAck.HomingAck := FALSE;
					uiHomingState := STATE_HOMING_FINISHED;
					IF SetupMode.Homing = FALSE THEN
		  		// Input was removed. Switch back to ModeAH. 	
		  		bHomingRemovedBeforeFinished := TRUE;	
					END_IF
        END_IF // end of 'IF (SetupMode.Homing = TRUE) AND (bHomingOld = FALSE) THEN'

    STATE_HOMING_INC_REAL_AXIS:
        // #####################################################################
				SetupModeAck.EnableAck  := TRUE; // Acknowledge SetupMode
    		// Homing for Real-Axis with incremental encoder
      	IF (SetupMode.Homing = TRUE) AND (bHomingOld = FALSE) THEN
       		// Set reference with incremental encoder
       		AdminCtrlExt._OpMode.en := ModeHoming;
    			enMyActAxisMode         := ModeHoming;
      	ELSIF AdminStatusExt.CmdDone AND AdminStatusExt.MODE_HOMING THEN
					// wait for Homing finished
					// Homing finished GOOD
					SetupModeAck.HomingAck := TRUE;
					uiHomingState := STATE_HOMING_FINISHED;
					IF SetupMode.Homing = FALSE THEN
		  		// Input was removed. Switch back to ModeAH. HomingAck stays active for one cycle... 	
		  		bHomingRemovedBeforeFinished := TRUE;	
					END_IF
      	ELSIF  DiagStatusExt.Error = TRUE AND SetupMode.Homing = FALSE THEN
					// wait for Homing finished BAD. Stay here untill the Homing is removed
					SetupModeAck.HomingAck := FALSE;
					uiHomingState := STATE_HOMING_FINISHED;
  	    // Input was removed. Switch back to ModeAH. 	
					bHomingRemovedBeforeFinished := TRUE;	
      	END_IF // end of 'IF (SetupMode.Homing = TRUE) AND (bHomingOld = FALSE) THEN'		
   
  STATE_HOMING_FINISHED:	
        // #####################################################################  
      	IF( ((SetupMode.Homing = FALSE) AND (bHomingOld = TRUE)) OR 
            (bHomingRemovedBeforeFinished = TRUE)                   ) THEN
					// falling edge on Homing or Homing removed before finished, reset to previous settings   
					AdminCtrlExt.SetAbsRef := FALSE;
        	AdminCtrlExt._OpMode.en := ModeAH;
					enMyActAxisMode         := ModeAH;
					// remove Acknowledge
					SetupModeAck.HomingAck := FALSE;
					bHomingRemovedBeforeFinished := FALSE;
					// wait for the next rising edge on Homing input
					IF AdminStatusExt.AxisFeatures.REAL_AXIS = TRUE THEN
						IF bAbsoluteEncoder = TRUE THEN
		      	  // absolute encoder
			  		  uiHomingState := STATE_HOMING_ABS_REAL_AXIS; // continue with homing an absolute real axis
		    	  ELSE
		      	  // incremental encoder
              uiHomingState := STATE_HOMING_INC_REAL_AXIS; // continue with homing an incremental real axis
						END_IF	
          ELSE 
		   		  uiHomingState := STATE_HOMING_VIRT_AXIS;   // continue with homing virtual axis
          END_IF
				END_IF	

    STATE_HOMING_NOT_POSSIBLE:
			SetupModeAck.EnableAck  := TRUE; // Acknowledge SetupMode
		  ; // nothing to do
      
    STATE_HOMING_NOT_IMPLEMENT:
			SetupModeAck.EnableAck  := TRUE; // Acknowledge SetupMode
		  IF( (SetupMode.Homing = TRUE) AND (bHomingOld = FALSE) ) THEN
        // signal an error, when user tries to home
   			SUPER^.mSetError( Error      := TRUE, 
       		                ErrorID    := INPUT_INVALID_ERROR, 
          	 	            ErrorIdent := HOMING_CONFIGURATION_ERR);
   			uiHomingState := STATE_HOMING_ERROR;   // continue with error
      END_IF
      
    STATE_HOMING_ERROR:
      // #####################################################################  
  		IF AdminCtrlExt.ClearError THEN
     		uiHomingState := STATE_HOMING_START;   // try a new start
  		END_IF	
	   

    ELSE 
        // #####################################################################  
   			// invalid state
   			SUPER^.mSetError( Error      := TRUE, 
       		              ErrorID    := STATE_MACHINE_ERROR, 
          	 	          ErrorIdent := HOMING_STATE_MACHINE_ERR);
   			uiHomingState := STATE_HOMING_ERROR;   // continue with error
	
    END_CASE // end of 'CASE uiHomingState OF'
  END_IF  // end of 'ELSIF SetupModeAck.SetupModeAck = TRUE THEN'
 
// Negative edge of Enable ? AND SetupMode was not aborted by assigning a new OpMode  
ELSIF bLatchSetupModeEnable AND bOriValuesStored = TRUE AND SetupModeAck.EnableAck = TRUE THEN
  // restore original values 
  VelModeCtrlExt.Velocity       := rOriVel;
  VelModeCtrlExt.Acceleration   := rOriAccel;
  AdminCtrlExt.StopDeceleration := rOriDecel;  // Defdb00116851 / Defdb00116875
  PosModeCtrlExt.Distance       := rOriDistance;
  PosModeCtrlExt.Velocity       := rOriVelPos;
  PosModeCtrlExt.Acceleration   := rOriAccelPos;
  PosModeCtrlExt.Deceleration   := rOriDecelPos;
  AdminCtrlExt._OpMode.en       := enOriAxisMode;
  bOriValuesStored              := FALSE;
  SetupModeAck.EnableAck        := FALSE; // remove acknowledge SetupMode
END_IF // SetupMode.Enable = TRUE

bLatchSetupModeEnable := SetupMode.Enable;
bHomingOld            := SetupMode.Homing;
END_ACTION

ACTION actSyncAccVel:
// Implements writing the Sync-Acceleration into parameter A-0-2791
// and writing the Sync-Velocity into parameter A-0-2790
// ####################################################
// Check if we are in bb. Otherwise we get errors.
// Do this only when sync is supported and the parameters are available.
// Distribute the load with using the axis address
IF AxisData[AdminCtrlExt.Axis.AxisNo].Axis_OperationMode = TRUE    AND 
   AdminStatusExt.AxisFeatures.OPMODE_SYNC = TRUE                   AND 
   (udiCycleCntInP4 > DINT_TO_UDINT(2 * AdminCtrlExt.Axis.AxisNo))     THEN 
  // write SyncAcceleration when changed 
  IF SyncModeCtrlExt.SyncAcceleration <> rLastSyncAcc OR bRestartSyncAcc THEN
    // changed value OR 1st time in Operation-Mode
    IF bExecWrSyncAcc = TRUE THEN
      // transmission is active, we need a new edge. Abort the actual transmission.
      bExecWrSyncAcc := FALSE;
    ELSE
      // no transmission active or we aborted the transmission, generate a new rising edge 
    bExecWrSyncAcc := TRUE;
    {IF defined (variable:InternalUsedSyncAcc)}
      // set Sync-Acceleration for Base-FB (needed for ML_Flexprofile inputs)
      InternalUsedSyncAcc:=ADR(SyncModeCtrlExt.SyncAcceleration);
    {END_IF}   
      // remember old value 
      rLastSyncAcc := SyncModeCtrlExt.SyncAcceleration;
      bRestartSyncAcc := FALSE;
  END_IF
    // start transmission 
    SyncModeStatusExt.SyncAccelerationDone := FALSE;
  END_IF
  IF fbWrSyncAcc.Done = TRUE THEN 
    // finished GOOD transmission 
    SyncModeStatusExt.SyncAccelerationDone := TRUE;
    bExecWrSyncAcc := FALSE;
  ELSIF fbWrSyncAcc.Error = TRUE THEN  
    // finished BAD transmission 
    bExecWrSyncAcc := FALSE;
    SUPER^.mSetError( Error      := TRUE, 
                      ErrorID    := fbWrSyncAcc.ErrorID, 
                      ErrorIdent := fbWrSyncAcc.ErrorIdent);
  END_IF  
  // call FB 
  fbWrSyncAcc(
	Execute:= bExecWrSyncAcc, 
	ParameterNumber:= FP_A_0_2791, 
	Value:= SyncModeCtrlExt.SyncAcceleration, 
	Axis:= AdminCtrlExt.Axis );	
	
  // ####################################################
  // write SyncVelocity when changed 
  IF SyncModeCtrlExt.SyncVelocity <> rLastSyncVel OR bRestartSyncVel THEN
    // changed value OR 1st time in Operation-Mode
    IF bExecWrSyncVel = TRUE THEN
      // transmission is active, we need a new edge. Abort the actual transmission.
      bExecWrSyncVel := FALSE;
    ELSE
      // no transmission active or we aborted the transmission, generate a new rising edge 
      bExecWrSyncVEl := TRUE;
    {IF defined (variable:InternalUsedSyncVelocity)}
      // set Sync-Velocity for Base-FB (needed for ML_Flexprofile inputs)
      InternalUsedSyncVelocity:=ADR(SyncModeCtrlExt.SyncVelocity);
    {END_IF}    
      // remember old value 
      rLastSyncVel := SyncModeCtrlExt.SyncVelocity;
      bRestartSyncVel := FALSE;
  END_IF
    // start transmission 
    SyncModeStatusExt.SyncVelocityDone := FALSE;
  END_IF
  IF fbWrSyncVel.Done = TRUE THEN 
    // finished GOOD transmission 
    SyncModeStatusExt.SyncVelocityDone := TRUE;
    bExecWrSyncVel := FALSE;
  ELSIF fbWrSyncVel.Error = TRUE THEN  
    // finished BAD transmission 
    bExecWrSyncVel := FALSE;
    SUPER^.mSetError( Error      := TRUE, 
                      ErrorID    := fbWrSyncVel.ErrorID, 
                      ErrorIdent := fbWrSyncVel.ErrorIdent);
  END_IF  
  // call FB 
  fbWrSyncVel(
	Execute:= bExecWrSyncVel, 
	ParameterNumber:= FP_A_0_2790, 
	Value:= SyncModeCtrlExt.SyncVelocity, 
	Axis:= AdminCtrlExt.Axis );	
ELSE
  // reset FBs when not in bb 
  fbWrSyncAcc( Execute:= FALSE,	Axis:= AdminCtrlExt.Axis );	
  fbWrSyncVel( Execute:= FALSE,	Axis:= AdminCtrlExt.Axis );	
END_IF
END_ACTION

METHOD mClearError : BOOL
VAR_INPUT
	boClearError : BOOL;
END_VAR
VAR
END_VAR
IF ADR(AdminCtrlExt) <> 0 THEN // check if the references are set (not needed, when references are set in FB_Init)
  AdminCtrlExt.ClearError := boClearError;
END_IF
IF ADR(DiagStatusExt) <> 0 THEN // check if the references are set (not needed, when references are set in FB_Init)
  mClearError := DiagStatusExt.Error;
END_IF
END_METHOD

METHOD mGetOpMode : MB_AXIS_MODE
VAR_INPUT
END_VAR
VAR
END_VAR
IF ADR(AdminStatusExt) <> 0 THEN // check if the references are set (not needed, when references are set in FB_Init)
  mGetOpMode := AdminStatusExt._OpModeAck;
END_IF
END_METHOD

METHOD mInitExtension
VAR_INPUT
	index: UINT;
END_VAR
VAR
END_VAR
SUPER^.mInitExtension(index);

// User: Assigment of user defined axis interface inputs
SetupMode  REF= arAxisCtrl_gb[index].SetupMode;

// User: Assigment of user defined axis interface outputs
SetupModeAck REF= arAxisStatus_gb[index].SetupMode;
AxisData_HMI REF= arAxisStatus_gb[index].AxisData_HMI;

// =================================================================
// Do not touch the following lines
// =================================================================

// Set the references for the AxisInterface FB 
AdminCtrlExt   	  REF= arAxisCtrl_gb[index].Admin;
PosModeCtrlExt    REF= arAxisCtrl_gb[index].PosMode;
VelModeCtrlExt    REF= arAxisCtrl_gb[index].VelMode;
SyncModeCtrlExt   REF= arAxisCtrl_gb[index].SyncMode;
TorqueModeCtrlExt REF= arAxisCtrl_gb[index].TorqueMode;
AdminStatusExt    REF= arAxisStatus_gb[index].Admin;
DiagStatusExt     REF= arAxisStatus_gb[index].Diag;
PosStatusExt      REF= arAxisStatus_gb[index].PosMode;
VelStatusExt      REF= arAxisStatus_gb[index].VelMode;
SyncModeStatusExt REF= arAxisStatus_gb[index].SyncMode;
// System: assign references of axis interface refresh FB
AdminCtrl 				REF= arAxisCtrl_gb[index].Admin;
PosModeCtrl 			REF= arAxisCtrl_gb[index].PosMode;
VelModeCtrl 			REF= arAxisCtrl_gb[index].VelMode;
SyncModeCtrl 			REF= arAxisCtrl_gb[index].SyncMode;
TorqueModeCtrl 		REF= arAxisCtrl_gb[index].TorqueMode;
AdminStatus 			REF= arAxisStatus_gb[index].Admin;
DiagStatus 				REF= arAxisStatus_gb[index].Diag;
PosStatus 				REF= arAxisStatus_gb[index].PosMode;
VelStatus 				REF= arAxisStatus_gb[index].VelMode;
SyncModeStatus 		REF= arAxisStatus_gb[index].SyncMode;
END_METHOD

METHOD mSetOpMode : MB_AXIS_MODE
VAR_INPUT
	enOpMode: MB_AXIS_MODE;
END_VAR
VAR
END_VAR
IF ADR(AdminCtrlExt) <> 0 THEN // check if the references are set (not needed, when references are set in FB_Init)
  AdminCtrlExt._OpMode.en := enOpMode;
END_IF
IF ADR(AdminStatusExt) <> 0 THEN // check if the references are set (not needed, when references are set in FB_Init)
  mSetOpMode := AdminStatusExt._OpModeAck;
END_IF
END_METHOD

END_FUNCTION_BLOCK

// IndraMotionMlc1/Application/POUs/AutoStow/P_AutoStow
PROGRAM P_AutoStow
VAR
	b_inc_timer: BOOL;
	r_autostow_counter: INT;
END_VAR


(* Functional Description 
The Autostow program will have a time that resets on the following conditions: 
	1. User Takes Authority : HHP,LMC or EGUI
	2. Locked State Estop, 
    3. Lockout switch Az/El (FI may be locked out at feed but the rest of the system is working)
    4. Pedestal door open 
    5. PSC door open
    6. Command sent 
     
Timer starts when all the conditions below are satisfied:
	1. Not in Locked State
	2. The counter starts immediatelly when no authority, time-out is 5minutes (default as per spec, but configurable). 
	3. The counter starts immediatelly when no connection, time-out is 5minutes (default as per spec, but configurable).
	4. The Pedestal and PSC doors are closed.
 
Autostow sequence: Various detail options can work, suggest we get details from MeerKAT & MK+ and try to be as consistant as possible. I will ask
1.	After timer has run out Sound horn for 5 seconds. 
2.	Wait TBC seconds. 
3.	Sound Horn and Stow.       

This task can be run at a 1 minute cadence   
*)


CASE CommandArbiter.Status.DscCmdAuthority OF
	 DscCmdAuthorityType.NoAuthority: b_inc_timer:= TRUE;
ELSE 
	 b_inc_timer:= FALSE; 
END_CASE 


// Check doors.  
IF CommandArbiter.Status.DscCmdAuthority = DscCmdAuthorityType.NoAuthority THEN
	IF b_DSDoor_Estop  OR b_PSCDoor_Estop THEN 
    	b_inc_timer:= FALSE; 
	ELSE // Command Authority
		CASE Management.Status.DscState OF 
     		DSCstatetype.Locked:  b_inc_timer:= FALSE; 
			DSCstatetype.Locked_Stowed: b_inc_timer:= FALSE;
			DSCstatetype.Stowed: b_inc_timer:= FALSE;
		ELSE 	 
			b_inc_timer:= TRUE;
		END_CASE
	END_IF
ELSE 
	b_inc_timer:= FALSE;
END_IF

IF b_inc_timer THEN 
	r_autostow_counter:=r_autostow_counter+1;
ELSE
   	r_autostow_counter:=0;
End_IF

IF r_autostow_counter >= gc_i_autostow_counter_max THEN 
   	b_activate_Az:=1;
	b_activate_El:=1;
    b_stow:=1; 
	r_goto_Az := 0;
	r_goto_El := 90;
	r_autostow_counter:=0;
	b_inc_timer:= FALSE;
END_IF

END_PROGRAM

